LIN {X 0,Y 99.884,Z 820.994,A -85,B 0,C 180,E1 25333.007,E2 25333.007} C_VEL
LIN {X 0,Y 124.493,Z 808.852,A -85,B 0,C 180,E1 25348.353,E2 25348.353} C_VEL
LIN {X 0,Y 153.117,Z 791.255,A -85,B 0,C 180,E1 25357.972,E2 25357.972} C_VEL
LIN {X 0,Y 182.881,Z 767.638,A -85,B 0,C 180,E1 25364.239,E2 25364.239} C_VEL
LIN {X 0,Y 189.802,Z 761.231,A -85,B 0,C 180,E1 25365.397,E2 25365.397} C_VEL
LIN {X 0,Y 195.132,Z 755.346,A -85,B 0,C 180,E1 25367.364,E2 25367.364} C_VEL
LIN {X 0,Y 198.666,Z 750.355,A -85,B 0,C 180,E1 25371.032,E2 25371.032} C_VEL
LIN {X 0,Y 200.372,Z 747.755,A -85,B 0,C 180,E1 25375.668,E2 25375.668} C_VEL
LIN {X 0,Y 200.976,Z 747.527,A -85,B 0,C 180,E1 25380.001,E2 25380.001} C_VEL
LIN {X 0,Y 199.237,Z 751.38,A -85,B 0,C 180,E1 25385.39,E2 25385.39} C_VEL
LIN {X 0,Y 197.973,Z 753.101,A -85,B 0,C 180,E1 25386.177,E2 25386.177} C_VEL
LIN {X 0,Y 169.301,Z 779.906,A -85,B 0,C 180,E1 25390.356,E2 25390.356} C_VEL
LIN {X 0,Y 138.614,Z 802.307,A -85,B 0,C 180,E1 25397.113,E2 25397.113} C_VEL
LIN {X 0,Y 110.818,Z 818.489,A -85,B 0,C 180,E1 25407.373,E2 25407.373} C_VEL
LIN {X 0,Y 86.48,Z 830.411,A -85,B 0,C 180,E1 25425.552,E2 25425.552} C_VEL
LIN {X 0,Y 75.414,Z 835.837,A -85,B 0,C 180,E1 25446.328,E2 25446.328} C_VEL
LIN {X 0,Y 73.158,Z 837.803,A -85,B 0,C 180,E1 25470.002,E2 25470.002} C_VEL
LIN {X 0,Y 75.424,Z 835.865,A -85,B 0,C 180,E1 25493.673,E2 25493.673} C_VEL
LIN {X 0,Y 91.541,Z 828.062,A -85,B 0,C 180,E1 25519.694,E2 25519.694} C_VEL
LIN {X 0,Y 116.651,Z 815.401,A -85,B 0,C 180,E1 25535.309,E2 25535.309} C_VEL
LIN {X 0,Y 147.138,Z 796.73,A -85,B 0,C 180,E1 25545.104,E2 25545.104} C_VEL
LIN {X 0,Y 177.618,Z 773.044,A -85,B 0,C 180,E1 25551.026,E2 25551.026} C_VEL
LIN {X 0,Y 197.983,Z 753.354,A -85,B 0,C 180,E1 25553.813,E2 25553.813} C_VEL
LIN {X 0,Y 199.783,Z 750.548,A -85,B 0,C 180,E1 25555.653,E2 25555.653} C_VEL
LIN {X 0,Y 201.058,Z 747.717,A -85,B 0,C 180,E1 25559.999,E2 25559.999} C_VEL
LIN {X 0,Y 200.407,Z 748.005,A -85,B 0,C 180,E1 25564.332,E2 25564.332} C_VEL
LIN {X 0,Y 197.938,Z 751.928,A -85,B 0,C 180,E1 25570.415,E2 25570.415} C_VEL
LIN {X 0,Y 193.785,Z 756.272,A -85,B 0,C 180,E1 25571.361,E2 25571.361} C_VEL
LIN {X 0,Y 164.984,Z 781.309,A -85,B 0,C 180,E1 25575.978,E2 25575.978} C_VEL
LIN {X 0,Y 134.949,Z 801.449,A -85,B 0,C 180,E1 25583.231,E2 25583.231} C_VEL
LIN {X 0,Y 105.987,Z 816.488,A -85,B 0,C 180,E1 25595.339,E2 25595.339} C_VEL
LIN {X 0,Y 82.666,Z 826.048,A -85,B 0,C 180,E1 25616.668,E2 25616.668} C_VEL
LIN {X 0,Y 74.295,Z 829.174,A -85,B 0,C 180,E1 25638.239,E2 25638.239} C_VEL
LIN {X 0,Y 73.683,Z 829.562,A -85,B 0,C 180,E1 25649.998,E2 25649.998} C_VEL
LIN {X 0,Y 77.339,Z 827.963,A -85,B 0,C 180,E1 25673.048,E2 25673.048} C_VEL
LIN {X 0,Y 94.189,Z 821.445,A -85,B 0,C 180,E1 25696.33,E2 25696.33} C_VEL
LIN {X 0,Y 120.489,Z 809.306,A -85,B 0,C 180,E1 25711.593,E2 25711.593} C_VEL
LIN {X 0,Y 150.297,Z 791.716,A -85,B 0,C 180,E1 25720.803,E2 25720.803} C_VEL
LIN {X 0,Y 180.886,Z 768.123,A -85,B 0,C 180,E1 25726.661,E2 25726.661} C_VEL
LIN {X 0,Y 197.67,Z 752.007,A -85,B 0,C 180,E1 25729.325,E2 25729.325} C_VEL
LIN {X 0,Y 198.666,Z 750.355,A -85,B 0,C 180,E1 25731.032,E2 25731.032} C_VEL
LIN {X 0,Y 198.812,Z 749.478,A -85,B 0,C 180,E1 25734.15,E2 25734.15} C_VEL
LIN {X 0,Y 194.974,Z 753.929,A -85,B 0,C 180,E1 25741.229,E2 25741.229} C_VEL
LIN {X 0,Y 194.065,Z 755.858,A -85,B 0,C 180,E1 25743.982,E2 25743.982} C_VEL
LIN {X 0,Y 163.979,Z 782.599,A -85,B 0,C 180,E1 25748.268,E2 25748.268} C_VEL
LIN {X 0,Y 133.056,Z 803.862,A -85,B 0,C 180,E1 25754.716,E2 25754.716} C_VEL
LIN {X 0,Y 104.295,Z 819.434,A -85,B 0,C 180,E1 25764.867,E2 25764.867} C_VEL
LIN {X 0,Y 80.849,Z 829.952,A -85,B 0,C 180,E1 25781.493,E2 25781.493} C_VEL
LIN {X 0,Y 68.087,Z 835.382,A -85,B 0,C 180,E1 25803.596,E2 25803.596} C_VEL
LIN {X 0,Y 65.227,Z 837.358,A -85,B 0,C 180,E1 25830.002,E2 25830.002} C_VEL
LIN {X 0,Y 68.642,Z 835.155,A -85,B 0,C 180,E1 25858.083,E2 25858.083} C_VEL
LIN {X 0,Y 86.807,Z 827.462,A -85,B 0,C 180,E1 25884.111,E2 25884.111} C_VEL
LIN {X 0,Y 115.581,Z 813.857,A -85,B 0,C 180,E1 25899.888,E2 25899.888} C_VEL
LIN {X 0,Y 148.967,Z 793.752,A -85,B 0,C 180,E1 25909.005,E2 25909.005} C_VEL
LIN {X 0,Y 178.898,Z 770.432,A -85,B 0,C 180,E1 25913.957,E2 25913.957} C_VEL
LIN {X 0,Y 194.078,Z 756.16,A -85,B 0,C 180,E1 25915.86,E2 25915.86} C_VEL
LIN {X 0,Y 195.432,Z 753.425,A -85,B 0,C 180,E1 25919.999,E2 25919.999} C_VEL
LIN {X 0,Y 194.735,Z 753.771,A -85,B 0,C 180,E1 25924.458,E2 25924.458} C_VEL
LIN {X 0,Y 193.418,Z 755.527,A -85,B 0,C 180,E1 25927.98,E2 25927.98} C_VEL
LIN {X 0,Y 192.198,Z 756.934,A -85,B 0,C 180,E1 25929.063,E2 25929.063} C_VEL
LIN {X 0,Y 162.977,Z 781.775,A -85,B 0,C 180,E1 25933.293,E2 25933.293} C_VEL
LIN {X 0,Y 132.746,Z 801.47,A -85,B 0,C 180,E1 25939.833,E2 25939.833} C_VEL
LIN {X 0,Y 103.062,Z 816.261,A -85,B 0,C 180,E1 25950.873,E2 25950.873} C_VEL
LIN {X 0,Y 77.793,Z 825.982,A -85,B 0,C 180,E1 25971.115,E2 25971.115} C_VEL
LIN {X 0,Y 66.554,Z 829.618,A -85,B 0,C 180,E1 25996.848,E2 25996.848} C_VEL
LIN {X 0,Y 65.782,Z 830.006,A -85,B 0,C 180,E1 26009.998,E2 26009.998} C_VEL
LIN {X 0,Y 70.094,Z 828.41,A -85,B 0,C 180,E1 26035.592,E2 26035.592} C_VEL
LIN {X 0,Y 84.222,Z 823.666,A -85,B 0,C 180,E1 26055.975,E2 26055.975} C_VEL
LIN {X 0,Y 110.809,Z 812.725,A -85,B 0,C 180,E1 26072.637,E2 26072.637} C_VEL
LIN {X 0,Y 139.683,Z 797.315,A -85,B 0,C 180,E1 26081.877,E2 26081.877} C_VEL
LIN {X 0,Y 170.365,Z 775.928,A -85,B 0,C 180,E1 26087.84,E2 26087.84} C_VEL
LIN {X 0,Y 192.711,Z 756.183,A -85,B 0,C 180,E1 26090.961,E2 26090.961} C_VEL
LIN {X 0,Y 194.716,Z 753.505,A -85,B 0,C 180,E1 26095.541,E2 26095.541} C_VEL
LIN {X 0,Y 195.349,Z 753.236,A -85,B 0,C 180,E1 26100.001,E2 26100.001} C_VEL
LIN {X 0,Y 194.974,Z 753.929,A -85,B 0,C 180,E1 26101.229,E2 26101.229} C_VEL
LIN {X 0,Y 192.253,Z 756.976,A -85,B 0,C 180,E1 26102.508,E2 26102.508} C_VEL
LIN {X 0,Y 178.528,Z 769.454,A -85,B 0,C 180,E1 26103.404,E2 26103.404} C_VEL
LIN {X 0,Y 147.135,Z 793.447,A -85,B 0,C 180,E1 26107.939,E2 26107.939} C_VEL
LIN {X 0,Y 113.771,Z 812.934,A -85,B 0,C 180,E1 26115.967,E2 26115.967} C_VEL
LIN {X 0,Y 83.388,Z 826.508,A -85,B 0,C 180,E1 26130.412,E2 26130.412} C_VEL
LIN {X 0,Y 63.672,Z 833.955,A -85,B 0,C 180,E1 26153.528,E2 26153.528} C_VEL
LIN {X 0,Y 57.593,Z 836.355,A -85,B 0,C 180,E1 26174.761,E2 26174.761} C_VEL
LIN {X 0,Y 57.315,Z 836.914,A -85,B 0,C 180,E1 26190.003,E2 26190.003} C_VEL
LIN {X 0,Y 60.982,Z 834.96,A -85,B 0,C 180,E1 26219.775,E2 26219.775} C_VEL
LIN {X 0,Y 80.731,Z 827.598,A -85,B 0,C 180,E1 26247.563,E2 26247.563} C_VEL
LIN {X 0,Y 110.792,Z 814.475,A -85,B 0,C 180,E1 26263.063,E2 26263.063} C_VEL
LIN {X 0,Y 145.353,Z 794.817,A -85,B 0,C 180,E1 26271.721,E2 26271.721} C_VEL
LIN {X 0,Y 178.223,Z 769.94,A -85,B 0,C 180,E1 26276.57,E2 26276.57} C_VEL
LIN {X 0,Y 188.15,Z 760.95,A -85,B 0,C 180,E1 26277.649,E2 26277.649} C_VEL
LIN {X 0,Y 189.628,Z 758.959,A -85,B 0,C 180,E1 26279.999,E2 26279.999} C_VEL
LIN {X 0,Y 188.288,Z 759.942,A -85,B 0,C 180,E1 26286.01,E2 26286.01} C_VEL
LIN {X 0,Y 187.946,Z 760.382,A -85,B 0,C 180,E1 26286.89,E2 26286.89} C_VEL
LIN {X 0,Y 158.206,Z 784.528,A -85,B 0,C 180,E1 26291.033,E2 26291.033} C_VEL
LIN {X 0,Y 126.907,Z 803.793,A -85,B 0,C 180,E1 26297.359,E2 26297.359} C_VEL
LIN {X 0,Y 97.209,Z 817.544,A -85,B 0,C 180,E1 26307.852,E2 26307.852} C_VEL
LIN {X 0,Y 69.899,Z 826.939,A -85,B 0,C 180,E1 26329.469,E2 26329.469} C_VEL
LIN {X 0,Y 58.861,Z 830.063,A -85,B 0,C 180,E1 26355.092,E2 26355.092} C_VEL
LIN {X 0,Y 57.899,Z 830.448,A -85,B 0,C 180,E1 26369.997,E2 26369.997} C_VEL
LIN {X 0,Y 63.019,Z 828.857,A -85,B 0,C 180,E1 26398.716,E2 26398.716} C_VEL
LIN {X 0,Y 78.876,Z 824.114,A -85,B 0,C 180,E1 26420.155,E2 26420.155} C_VEL
LIN {X 0,Y 107.374,Z 813.178,A -85,B 0,C 180,E1 26436.422,E2 26436.422} C_VEL
LIN {X 0,Y 138.883,Z 796.875,A -85,B 0,C 180,E1 26445.352,E2 26445.352} C_VEL
LIN {X 0,Y 170.667,Z 774.971,A -85,B 0,C 180,E1 26450.723,E2 26450.723} C_VEL
LIN {X 0,Y 187.837,Z 760.224,A -85,B 0,C 180,E1 26453.064,E2 26453.064} C_VEL
LIN {X 0,Y 188.833,Z 759.063,A -85,B 0,C 180,E1 26455.402,E2 26455.402} C_VEL
LIN {X 0,Y 189.277,Z 759.221,A -85,B 0,C 180,E1 26460.822,E2 26460.822} C_VEL
LIN {X 0,Y 188.874,Z 759.929,A -85,B 0,C 180,E1 26462.014,E2 26462.014} C_VEL
LIN {X 0,Y 178.528,Z 769.454,A -85,B 0,C 180,E1 26463.404,E2 26463.404} C_VEL
LIN {X 0,Y 164.754,Z 780.338,A -85,B 0,C 180,E1 26463.71,E2 26463.71} C_VEL
LIN {X 0,Y 150.338,Z 790.211,A -85,B 0,C 180,E1 26464.149,E2 26464.149} C_VEL
LIN {X 0,Y 118.789,Z 808.908,A -85,B 0,C 180,E1 26470.089,E2 26470.089} C_VEL
LIN {X 0,Y 86.351,Z 823.488,A -85,B 0,C 180,E1 26481.504,E2 26481.504} C_VEL
LIN {X 0,Y 61.326,Z 832.18,A -85,B 0,C 180,E1 26502.216,E2 26502.216} C_VEL
LIN {X 0,Y 49.906,Z 835.905,A -85,B 0,C 180,E1 26532.343,E2 26532.343} C_VEL
LIN {X 0,Y 49.374,Z 836.468,A -85,B 0,C 180,E1 26550.003,E2 26550.003} C_VEL
LIN {X 0,Y 54.102,Z 834.506,A -85,B 0,C 180,E1 26584.039,E2 26584.039} C_VEL
LIN {X 0,Y 76.643,Z 827.139,A -85,B 0,C 180,E1 26612.748,E2 26612.748} C_VEL
LIN {X 0,Y 108.684,Z 814.011,A -85,B 0,C 180,E1 26627.207,E2 26627.207} C_VEL
LIN {X 0,Y 144.395,Z 794.344,A -85,B 0,C 180,E1 26634.963,E2 26634.963} C_VEL
LIN {X 0,Y 177.921,Z 769.447,A -85,B 0,C 180,E1 26639.192,E2 26639.192} C_VEL
LIN {X 0,Y 183.698,Z 764.39,A -85,B 0,C 180,E1 26639.999,E2 26639.999} C_VEL
LIN {X 0,Y 182.421,Z 765.109,A -85,B 0,C 180,E1 26645.136,E2 26645.136} C_VEL
LIN {X 0,Y 151.362,Z 788.656,A -85,B 0,C 180,E1 26648.958,E2 26648.958} C_VEL
LIN {X 0,Y 119.97,Z 806.58,A -85,B 0,C 180,E1 26654.969,E2 26654.969} C_VEL
LIN {X 0,Y 89.506,Z 819.481,A -85,B 0,C 180,E1 26665.441,E2 26665.441} C_VEL
LIN {X 0,Y 63.06,Z 827.637,A -85,B 0,C 180,E1 26686.07,E2 26686.07} C_VEL
LIN {X 0,Y 51.239,Z 830.508,A -85,B 0,C 180,E1 26712.81,E2 26712.81} C_VEL
LIN {X 0,Y 49.995,Z 830.892,A -85,B 0,C 180,E1 26729.997,E2 26729.997} C_VEL
LIN {X 0,Y 56.175,Z 829.304,A -85,B 0,C 180,E1 26762.615,E2 26762.615} C_VEL
LIN {X 0,Y 79.545,Z 822.796,A -85,B 0,C 180,E1 26788.924,E2 26788.924} C_VEL
LIN {X 0,Y 111.095,Z 810.662,A -85,B 0,C 180,E1 26802.547,E2 26802.547} C_VEL
LIN {X 0,Y 144.205,Z 793.094,A -85,B 0,C 180,E1 26809.831,E2 26809.831} C_VEL
LIN {X 0,Y 176.909,Z 769.579,A -85,B 0,C 180,E1 26814.206,E2 26814.206} C_VEL
LIN {X 0,Y 182.434,Z 764.862,A -85,B 0,C 180,E1 26814.8,E2 26814.8} C_VEL
LIN {X 0,Y 183.63,Z 764.22,A -85,B 0,C 180,E1 26820.001,E2 26820.001} C_VEL
LIN {X 0,Y 154.352,Z 787.527,A -85,B 0,C 180,E1 26823.593,E2 26823.593} C_VEL
LIN {X 0,Y 150.338,Z 790.211,A -85,B 0,C 180,E1 26824.149,E2 26824.149} C_VEL
LIN {X 0,Y 135.405,Z 799.256,A -85,B 0,C 180,E1 26824.822,E2 26824.822} C_VEL
LIN {X 0,Y 119.946,Z 807.298,A -85,B 0,C 180,E1 26825.703,E2 26825.703} C_VEL
LIN {X 0,Y 87.793,Z 821.536,A -85,B 0,C 180,E1 26834.544,E2 26834.544} C_VEL
LIN {X 0,Y 56.17,Z 831.722,A -85,B 0,C 180,E1 26856.041,E2 26856.041} C_VEL
LIN {X 0,Y 42.343,Z 835.455,A -85,B 0,C 180,E1 26889.053,E2 26889.053} C_VEL
LIN {X 0,Y 41.429,Z 836.022,A -85,B 0,C 180,E1 26910.004,E2 26910.004} C_VEL
LIN {X 0,Y 47.607,Z 834.052,A -85,B 0,C 180,E1 26949.503,E2 26949.503} C_VEL
LIN {X 0,Y 73.26,Z 826.68,A -85,B 0,C 180,E1 26978.441,E2 26978.441} C_VEL
LIN {X 0,Y 107.169,Z 813.551,A -85,B 0,C 180,E1 26991.48,E2 26991.48} C_VEL
LIN {X 0,Y 143.908,Z 793.875,A -85,B 0,C 180,E1 26998.211,E2 26998.211} C_VEL
LIN {X 0,Y 177.143,Z 769.661,A -85,B 0,C 180,E1 27001.946,E2 27001.946} C_VEL
LIN {X 0,Y 176.977,Z 769.732,A -85,B 0,C 180,E1 27002.843,E2 27002.843} C_VEL
LIN {X 0,Y 146.656,Z 791.472,A -85,B 0,C 180,E1 27006.441,E2 27006.441} C_VEL
LIN {X 0,Y 111.616,Z 810.098,A -85,B 0,C 180,E1 27012.672,E2 27012.672} C_VEL
LIN {X 0,Y 81.99,Z 821.425,A -85,B 0,C 180,E1 27022.58,E2 27022.58} C_VEL
LIN {X 0,Y 58.698,Z 827.831,A -85,B 0,C 180,E1 27039.298,E2 27039.298} C_VEL
LIN {X 0,Y 43.725,Z 830.953,A -85,B 0,C 180,E1 27069.737,E2 27069.737} C_VEL
LIN {X 0,Y 42.117,Z 831.334,A -85,B 0,C 180,E1 27089.996,E2 27089.996} C_VEL
LIN {X 0,Y 49.663,Z 829.75,A -85,B 0,C 180,E1 27127.566,E2 27127.566} C_VEL
LIN {X 0,Y 75.728,Z 823.244,A -85,B 0,C 180,E1 27154.113,E2 27154.113} C_VEL
LIN {X 0,Y 108.963,Z 811.114,A -85,B 0,C 180,E1 27166.564,E2 27166.564} C_VEL
LIN {X 0,Y 143.013,Z 793.554,A -85,B 0,C 180,E1 27172.974,E2 27172.974} C_VEL
LIN {X 0,Y 176.924,Z 769.531,A -85,B 0,C 180,E1 27176.935,E2 27176.935} C_VEL
LIN {X 0,Y 177.12,Z 769.448,A -85,B 0,C 180,E1 27178.061,E2 27178.061} C_VEL
LIN {X 0,Y 145.778,Z 792.49,A -85,B 0,C 180,E1 27181.55,E2 27181.55} C_VEL
LIN {X 0,Y 119.946,Z 807.298,A -85,B 0,C 180,E1 27185.703,E2 27185.703} C_VEL
LIN {X 0,Y 104.006,Z 814.363,A -85,B 0,C 180,E1 27186.888,E2 27186.888} C_VEL
LIN {X 0,Y 87.86,Z 820.433,A -85,B 0,C 180,E1 27188.679,E2 27188.679} C_VEL
LIN {X 0,Y 55.766,Z 830.347,A -85,B 0,C 180,E1 27205.007,E2 27205.007} C_VEL
LIN {X 0,Y 34.963,Z 835.004,A -85,B 0,C 180,E1 27244.344,E2 27244.344} C_VEL
LIN {X 0,Y 33.48,Z 835.576,A -85,B 0,C 180,E1 27270.005,E2 27270.005} C_VEL
LIN {X 0,Y 41.673,Z 833.597,A -85,B 0,C 180,E1 27316.611,E2 27316.611} C_VEL
LIN {X 0,Y 70.665,Z 826.221,A -85,B 0,C 180,E1 27344.623,E2 27344.623} C_VEL
LIN {X 0,Y 106.266,Z 813.092,A -85,B 0,C 180,E1 27355.845,E2 27355.845} C_VEL
LIN {X 0,Y 141.98,Z 794.533,A -85,B 0,C 180,E1 27361.264,E2 27361.264} C_VEL
LIN {X 0,Y 151.522,Z 788.479,A -85,B 0,C 180,E1 27362.221,E2 27362.221} C_VEL
LIN {X 0,Y 151.58,Z 788.402,A -85,B 0,C 180,E1 27362.727,E2 27362.727} C_VEL
LIN {X 0,Y 117.97,Z 806.976,A -85,B 0,C 180,E1 27367.181,E2 27367.181} C_VEL
LIN {X 0,Y 84.722,Z 820.114,A -85,B 0,C 180,E1 27375.246,E2 27375.246} C_VEL
LIN {X 0,Y 54.003,Z 828.279,A -85,B 0,C 180,E1 27392.738,E2 27392.738} C_VEL
LIN {X 0,Y 36.387,Z 831.398,A -85,B 0,C 180,E1 27425.407,E2 27425.407} C_VEL
LIN {X 0,Y 34.211,Z 831.777,A -85,B 0,C 180,E1 27449.995,E2 27449.995} C_VEL
LIN {X 0,Y 49.061,Z 829.257,A -85,B 0,C 180,E1 27501.894,E2 27501.894} C_VEL
LIN {X 0,Y 79.278,Z 821.786,A -85,B 0,C 180,E1 27522.719,E2 27522.719} C_VEL
LIN {X 0,Y 115.625,Z 807.932,A -85,B 0,C 180,E1 27532.303,E2 27532.303} C_VEL
LIN {X 0,Y 149.716,Z 789.397,A -85,B 0,C 180,E1 27536.991,E2 27536.991} C_VEL
LIN {X 0,Y 151.587,Z 788.215,A -85,B 0,C 180,E1 27537.17,E2 27537.17} C_VEL
LIN {X 0,Y 151.517,Z 788.308,A -85,B 0,C 180,E1 27537.772,E2 27537.772} C_VEL
LIN {X 0,Y 117.415,Z 807.794,A -85,B 0,C 180,E1 27542.097,E2 27542.097} C_VEL
LIN {X 0,Y 87.86,Z 820.433,A -85,B 0,C 180,E1 27548.679,E2 27548.679} C_VEL
LIN {X 0,Y 71.428,Z 825.402,A -85,B 0,C 180,E1 27551.301,E2 27551.301} C_VEL
LIN {X 0,Y 54.972,Z 829.347,A -85,B 0,C 180,E1 27555.526,E2 27555.526} C_VEL
LIN {X 0,Y 36.572,Z 833.111,A -85,B 0,C 180,E1 27574.115,E2 27574.115} C_VEL
LIN {X 0,Y 25.543,Z 835.131,A -85,B 0,C 180,E1 27630.006,E2 27630.006} C_VEL
LIN {X 0,Y 36.578,Z 833.142,A -85,B 0,C 180,E1 27685.886,E2 27685.886} C_VEL
LIN {X 0,Y 68.944,Z 825.763,A -85,B 0,C 180,E1 27711.213,E2 27711.213} C_VEL
LIN {X 0,Y 105.988,Z 812.629,A -85,B 0,C 180,E1 27720.293,E2 27720.293} C_VEL
LIN {X 0,Y 121.232,Z 805.647,A -85,B 0,C 180,E1 27722.385,E2 27722.385} C_VEL
LIN {X 0,Y 121.271,Z 805.598,A -85,B 0,C 180,E1 27722.79,E2 27722.79} C_VEL
LIN {X 0,Y 84.506,Z 820.095,A -85,B 0,C 180,E1 27729.517,E2 27729.517} C_VEL
LIN {X 0,Y 50.132,Z 828.727,A -85,B 0,C 180,E1 27745.029,E2 27745.029} C_VEL
LIN {X 0,Y 29.359,Z 831.843,A -85,B 0,C 180,E1 27778.949,E2 27778.949} C_VEL
LIN {X 0,Y 26.303,Z 832.221,A -85,B 0,C 180,E1 27809.994,E2 27809.994} C_VEL
LIN {X 0,Y 38.312,Z 830.641,A -85,B 0,C 180,E1 27862.214,E2 27862.214} C_VEL
LIN {X 0,Y 70.232,Z 824.144,A -85,B 0,C 180,E1 27885.944,E2 27885.944} C_VEL
LIN {X 0,Y 106.392,Z 812.021,A -85,B 0,C 180,E1 27894.959,E2 27894.959} C_VEL
LIN {X 0,Y 121.272,Z 805.463,A -85,B 0,C 180,E1 27897.142,E2 27897.142} C_VEL
LIN {X 0,Y 121.225,Z 805.522,A -85,B 0,C 180,E1 27897.634,E2 27897.634} C_VEL
LIN {X 0,Y 84.902,Z 820.698,A -85,B 0,C 180,E1 27903.833,E2 27903.833} C_VEL
LIN {X 0,Y 54.972,Z 829.347,A -85,B 0,C 180,E1 27915.526,E2 27915.526} C_VEL
LIN {X 0,Y 42.942,Z 831.639,A -85,B 0,C 180,E1 27921.185,E2 27921.185} C_VEL
LIN {X 0,Y 24.915,Z 833.703,A -85,B 0,C 180,E1 27935.72,E2 27935.72} C_VEL
LIN {X 0,Y 23.407,Z 833.85,A -85,B 0,C 180,E1 27939.523,E2 27939.523} C_VEL
LIN {X 0,Y 17.584,Z 834.684,A -85,B 0,C 180,E1 27990.009,E2 27990.009} C_VEL
LIN {X 0,Y 32.734,Z 832.69,A -85,B 0,C 180,E1 28057.692,E2 28057.692} C_VEL
LIN {X 0,Y 68.175,Z 825.304,A -85,B 0,C 180,E1 28078.036,E2 28078.036} C_VEL
LIN {X 0,Y 90.951,Z 818.151,A -85,B 0,C 180,E1 28082.753,E2 28082.753} C_VEL
LIN {X 0,Y 54.308,Z 827.907,A -85,B 0,C 180,E1 28092.625,E2 28092.625} C_VEL
LIN {X 0,Y 22.93,Z 832.288,A -85,B 0,C 180,E1 28128.669,E2 28128.669} C_VEL
LIN {X 0,Y 18.395,Z 832.665,A -85,B 0,C 180,E1 28169.991,E2 28169.991} C_VEL
LIN {X 0,Y 36.281,Z 830.803,A -85,B 0,C 180,E1 28235.341,E2 28235.341} C_VEL
LIN {X 0,Y 68.729,Z 824.594,A -85,B 0,C 180,E1 28252.428,E2 28252.428} C_VEL
LIN {X 0,Y 90.942,Z 818.059,A -85,B 0,C 180,E1 28257.282,E2 28257.282} C_VEL
LIN {X 0,Y 51.361,Z 829.332,A -85,B 0,C 180,E1 28267.941,E2 28267.941} C_VEL
LIN {X 0,Y 23.407,Z 833.85,A -85,B 0,C 180,E1 28299.523,E2 28299.523} C_VEL
LIN {X 0,Y 14.939,Z 834.532,A -85,B 0,C 180,E1 28330.471,E2 28330.471} C_VEL
LIN {X 0,Y 18.051,Z 833.537,A -85,B 0,C 180,E1 28416.618,E2 28416.618} C_VEL
LIN {X 0,Y 46.964,Z 829.669,A -85,B 0,C 180,E1 28439.997,E2 28439.997} C_VEL
LIN {X 0,Y 56.525,Z 827.709,A -85,B 0,C 180,E1 28442.654,E2 28442.654} C_VEL
LIN {X 0,Y 31.206,Z 831.571,A -85,B 0,C 180,E1 28453.965,E2 28453.965} C_VEL
LIN {X 0,Y 10.496,Z 833.108,A -85,B 0,C 180,E1 28529.984,E2 28529.984} C_VEL
LIN {X 0,Y 31.212,Z 831.534,A -85,B 0,C 180,E1 28605.95,E2 28605.95} C_VEL
LIN {X 0,Y 56.649,Z 827.623,A -85,B 0,C 180,E1 28617.317,E2 28617.317} C_VEL
LIN {X 0,Y 30.581,Z 832.201,A -85,B 0,C 180,E1 28628.066,E2 28628.066} C_VEL
LIN {X 0,Y 9.643,Z 834.238,A -85,B 0,C 180,E1 28710.017,E2 28710.017} C_VEL
LIN {X 0,Y 18.051,Z 833.537,A -85,B 0,C 180,E1 28776.618,E2 28776.618} C_VEL
LIN {X 0,Y 14.146,Z 833.507,A -85,B 0,C 180,E1 28788.096,E2 28788.096} C_VEL
LIN {X 0,Y 2.205,Z 833.569,A -85,B 0,C 180,E1 28909.108,E2 28909.108} C_VEL
LIN {X 0,Y 5.438,Z 833.422,A -85,B 0,C 180,E1 28956.094,E2 28956.094} C_VEL
LIN {X 0,Y 15.204,Z 833.155,A -85,B 0,C 180,E1 28974.629,E2 28974.629} C_VEL
LIN {X 0,Y 1.672,Z 833.791,A -85,B 0,C 180,E1 29070.097,E2 29070.097} C_VEL
LIN {X 0,Y 15.204,Z 833.178,A -85,B 0,C 180,E1 29165.139,E2 29165.139} C_VEL
LIN {X 0,Y 5.438,Z 833.422,A -85,B 0,C 180,E1 29316.094,E2 29316.094} C_VEL
LIN {X 0,Y 7.31,Z 835.421,A -85,B 0,C 180,E1 29323.741,E2 29323.741} C_VEL
LIN {X 0,Y 7.31,Z 862.5,A -85,B 0,C 180,E1 29323.741,E2 29323.741} C_VEL
LIN {X 0,Y 7.31,Z 862.5,A -85,B 0,C 180,E1 29323.741,E2 29323.741}

QRS_NEXT_CUT()
PTP {E1 29336.868,E2 29336.868}
PTP {X 0,Y 607.922,A -85,B 0,C 180,E1 29336.868,E2 29336.868,E3 0,E4 0,E5 0,E6 0}
QRS_SPEED_INIT()
LIN {X 0,Y 607.922,Z 862.5,A -85,B 0,C 180,E1 29336.868,E2 29336.868,E3 0,E4 0,E5 0,E6 0} C_VEL
LIN {X 0,Y 607.922,Z 262.089,A -85,B 0,C 180,E1 29336.868,E2 29336.868} C_VEL
LIN {X 0,Y 607.922,Z 254.014,A -85,B 0,C 180,E1 29336.868,E2 29336.868} C_VEL
LIN {X 0,Y 607.917,Z 252.014,A -85,B 0,C 180,E1 29336.68,E2 29336.68} C_VEL
LIN {X 0,Y 607.854,Z 252.011,A -85,B 0,C 180,E1 29333.578,E2 29333.578} C_VEL
LIN {X 0,Y 607.917,Z 252.011,A -85,B 0,C 180,E1 29330.533,E2 29330.533} C_VEL
LIN {X 0,Y 607.86,Z 252.012,A -85,B 0,C 180,E1 29327.46,E2 29327.46} C_VEL
LIN {X 0,Y 607.916,Z 252.009,A -85,B 0,C 180,E1 29324.351,E2 29324.351} C_VEL
LIN {X 0,Y 607.875,Z 252.012,A -85,B 0,C 180,E1 29321.192,E2 29321.192} C_VEL
LIN {X 0,Y 607.901,Z 252.006,A -85,B 0,C 180,E1 29317.975,E2 29317.975} C_VEL
LIN {X 0,Y 607.907,Z 252.015,A -85,B 0,C 180,E1 29314.768,E2 29314.768} C_VEL
LIN {X 0,Y 607.885,Z 252.008,A -85,B 0,C 180,E1 29311.618,E2 29311.618} C_VEL
LIN {X 0,Y 607.912,Z 252.012,A -85,B 0,C 180,E1 29308.575,E2 29308.575} C_VEL
LIN {X 0,Y 607.886,Z 252.009,A -85,B 0,C 180,E1 29305.426,E2 29305.426} C_VEL
LIN {X 0,Y 607.905,Z 252.01,A -85,B 0,C 180,E1 29302.395,E2 29302.395} C_VEL
LIN {X 0,Y 607.891,Z 252.01,A -85,B 0,C 180,E1 29299.233,E2 29299.233} C_VEL
LIN {X 0,Y 607.902,Z 252.008,A -85,B 0,C 180,E1 29296.087,E2 29296.087} C_VEL
LIN {X 0,Y 607.904,Z 252.012,A -85,B 0,C 180,E1 29292.915,E2 29292.915} C_VEL
LIN {X 0,Y 607.91,Z 252.004,A -85,B 0,C 180,E1 29289.654,E2 29289.654} C_VEL
LIN {X 0,Y 607.899,Z 252.013,A -85,B 0,C 180,E1 29286.423,E2 29286.423} C_VEL
LIN {X 0,Y 607.903,Z 252.007,A -85,B 0,C 180,E1 29283.209,E2 29283.209} C_VEL
LIN {X 0,Y 607.908,Z 252.244,A -85,B 0,C 180,E1 29282.871,E2 29282.871} C_VEL
LIN {X 0,Y 607.916,Z 262.06,A -85,B 0,C 180,E1 29282.155,E2 29282.155} C_VEL
LIN {X 0,Y 607.91,Z 307.319,A -85,B 0,C 180,E1 29279.079,E2 29279.079} C_VEL
LIN {X 0,Y 607.915,Z 329.228,A -85,B 0,C 180,E1 29277.639,E2 29277.639} C_VEL
LIN {X 0,Y 607.906,Z 572.151,A -85,B 0,C 180,E1 29274.503,E2 29274.503} C_VEL
LIN {X 0,Y 607.916,Z 596.076,A -85,B 0,C 180,E1 29274.138,E2 29274.138} C_VEL
LIN {X 0,Y 607.907,Z 615.328,A -85,B 0,C 180,E1 29273.686,E2 29273.686} C_VEL
LIN {X 0,Y 607.906,Z 635.144,A -85,B 0,C 180,E1 29273.044,E2 29273.044} C_VEL
LIN {X 0,Y 607.914,Z 653.488,A -85,B 0,C 180,E1 29272.278,E2 29272.278} C_VEL
LIN {X 0,Y 607.918,Z 672.334,A -85,B 0,C 180,E1 29271.314,E2 29271.314} C_VEL
LIN {X 0,Y 607.918,Z 690.309,A -85,B 0,C 180,E1 29270.205,E2 29270.205} C_VEL
LIN {X 0,Y 607.912,Z 707.273,A -85,B 0,C 180,E1 29268.963,E2 29268.963} C_VEL
LIN {X 0,Y 607.916,Z 723.45,A -85,B 0,C 180,E1 29267.566,E2 29267.566} C_VEL
LIN {X 0,Y 607.913,Z 738.451,A -85,B 0,C 180,E1 29266.04,E2 29266.04} C_VEL
LIN {X 0,Y 607.916,Z 752.426,A -85,B 0,C 180,E1 29264.361,E2 29264.361} C_VEL
LIN {X 0,Y 607.912,Z 764.497,A -85,B 0,C 180,E1 29262.635,E2 29262.635} C_VEL
LIN {X 0,Y 607.904,Z 774.619,A -85,B 0,C 180,E1 29260.903,E2 29260.903} C_VEL
LIN {X 0,Y 607.912,Z 783.37,A -85,B 0,C 180,E1 29259.084,E2 29259.084} C_VEL
LIN {X 0,Y 607.907,Z 790.348,A -85,B 0,C 180,E1 29257.276,E2 29257.276} C_VEL
LIN {X 0,Y 607.903,Z 795.888,A -85,B 0,C 180,E1 29255.379,E2 29255.379} C_VEL
LIN {X 0,Y 607.901,Z 799.664,A -85,B 0,C 180,E1 29253.489,E2 29253.489} C_VEL
LIN {X 0,Y 607.903,Z 801.841,A -85,B 0,C 180,E1 29251.602,E2 29251.602} C_VEL
LIN {X 0,Y 607.904,Z 802.45,A -85,B 0,C 180,E1 29249.717,E2 29249.717} C_VEL
LIN {X 0,Y 607.911,Z 801.498,A -85,B 0,C 180,E1 29247.832,E2 29247.832} C_VEL
LIN {X 0,Y 607.913,Z 798.71,A -85,B 0,C 180,E1 29245.85,E2 29245.85} C_VEL
LIN {X 0,Y 607.919,Z 794.356,A -85,B 0,C 180,E1 29243.958,E2 29243.958} C_VEL
LIN {X 0,Y 607.915,Z 788.287,A -85,B 0,C 180,E1 29242.059,E2 29242.059} C_VEL
LIN {X 0,Y 607.91,Z 780.817,A -85,B 0,C 180,E1 29240.247,E2 29240.247} C_VEL
LIN {X 0,Y 607.904,Z 771.474,A -85,B 0,C 180,E1 29238.425,E2 29238.425} C_VEL
LIN {X 0,Y 607.912,Z 760.614,A -85,B 0,C 180,E1 29236.688,E2 29236.688} C_VEL
LIN {X 0,Y 607.91,Z 748.345,A -85,B 0,C 180,E1 29235.036,E2 29235.036} C_VEL
LIN {X 0,Y 607.916,Z 734.67,A -85,B 0,C 180,E1 29233.469,E2 29233.469} C_VEL
LIN {X 0,Y 607.912,Z 719.508,A -85,B 0,C 180,E1 29231.989,E2 29231.989} C_VEL
LIN {X 0,Y 607.918,Z 702.707,A -85,B 0,C 180,E1 29230.596,E2 29230.596} C_VEL
LIN {X 0,Y 607.918,Z 685.576,A -85,B 0,C 180,E1 29229.393,E2 29229.393} C_VEL
LIN {X 0,Y 607.918,Z 667.445,A -85,B 0,C 180,E1 29228.322,E2 29228.322} C_VEL
LIN {X 0,Y 607.918,Z 648.751,A -85,B 0,C 180,E1 29227.416,E2 29227.416} C_VEL
LIN {X 0,Y 607.915,Z 629.645,A -85,B 0,C 180,E1 29226.674,E2 29226.674} C_VEL
LIN {X 0,Y 607.906,Z 609.883,A -85,B 0,C 180,E1 29226.082,E2 29226.082} C_VEL
LIN {X 0,Y 607.913,Z 589.981,A -85,B 0,C 180,E1 29225.657,E2 29225.657} C_VEL
LIN {X 0,Y 607.914,Z 329.113,A -85,B 0,C 180,E1 29222.267,E2 29222.267} C_VEL
LIN {X 0,Y 607.918,Z 285.168,A -85,B 0,C 180,E1 29219.338,E2 29219.338} C_VEL
LIN {X 0,Y 607.911,Z 252.36,A -85,B 0,C 180,E1 29217.059,E2 29217.059} C_VEL
LIN {X 0,Y 607.919,Z 252.003,A -85,B 0,C 180,E1 29216.454,E2 29216.454} C_VEL
LIN {X 0,Y 607.912,Z 252.014,A -85,B 0,C 180,E1 29213.108,E2 29213.108} C_VEL
LIN {X 0,Y 607.895,Z 252.006,A -85,B 0,C 180,E1 29209.977,E2 29209.977} C_VEL
LIN {X 0,Y 607.9,Z 252.01,A -85,B 0,C 180,E1 29206.827,E2 29206.827} C_VEL
LIN {X 0,Y 607.896,Z 252.01,A -85,B 0,C 180,E1 29203.694,E2 29203.694} C_VEL
LIN {X 0,Y 607.897,Z 252.007,A -85,B 0,C 180,E1 29200.518,E2 29200.518} C_VEL
LIN {X 0,Y 607.907,Z 252.013,A -85,B 0,C 180,E1 29197.367,E2 29197.367} C_VEL
LIN {X 0,Y 607.914,Z 252.004,A -85,B 0,C 180,E1 29194.115,E2 29194.115} C_VEL
LIN {X 0,Y 607.89,Z 252.011,A -85,B 0,C 180,E1 29190.845,E2 29190.845} C_VEL
LIN {X 0,Y 607.909,Z 252.007,A -85,B 0,C 180,E1 29187.74,E2 29187.74} C_VEL
LIN {X 0,Y 607.879,Z 252.01,A -85,B 0,C 180,E1 29184.555,E2 29184.555} C_VEL
LIN {X 0,Y 607.912,Z 252.012,A -85,B 0,C 180,E1 29181.416,E2 29181.416} C_VEL
LIN {X 0,Y 607.876,Z 252.009,A -85,B 0,C 180,E1 29178.311,E2 29178.311} C_VEL
LIN {X 0,Y 607.899,Z 252.014,A -85,B 0,C 180,E1 29175.063,E2 29175.063} C_VEL
LIN {X 0,Y 607.887,Z 252.008,A -85,B 0,C 180,E1 29171.961,E2 29171.961} C_VEL
LIN {X 0,Y 607.867,Z 252.013,A -85,B 0,C 180,E1 29168.704,E2 29168.704} C_VEL
LIN {X 0,Y 607.91,Z 252.008,A -85,B 0,C 180,E1 29165.664,E2 29165.664} C_VEL
LIN {X 0,Y 607.855,Z 252.012,A -85,B 0,C 180,E1 29162.546,E2 29162.546} C_VEL
LIN {X 0,Y 607.912,Z 252.01,A -85,B 0,C 180,E1 29159.529,E2 29159.529} C_VEL
LIN {X 0,Y 607.845,Z 252.013,A -85,B 0,C 180,E1 29156.416,E2 29156.416} C_VEL
LIN {X 0,Y 607.911,Z 252.013,A -85,B 0,C 180,E1 29153.389,E2 29153.389} C_VEL
LIN {X 0,Y 607.835,Z 252.014,A -85,B 0,C 180,E1 29150.341,E2 29150.341} C_VEL
LIN {X 0,Y 607.918,Z 252.014,A -85,B 0,C 180,E1 29147.268,E2 29147.268} C_VEL
LIN {X 0,Y 607.826,Z 252.015,A -85,B 0,C 180,E1 29144.214,E2 29144.214} C_VEL
LIN {X 0,Y 607.906,Z 252.015,A -85,B 0,C 180,E1 29141.194,E2 29141.194} C_VEL
LIN {X 0,Y 607.835,Z 252.014,A -85,B 0,C 180,E1 29138.176,E2 29138.176} C_VEL
LIN {X 0,Y 607.919,Z 252.012,A -85,B 0,C 180,E1 29135.099,E2 29135.099} C_VEL
LIN {X 0,Y 607.845,Z 252.013,A -85,B 0,C 180,E1 29132.043,E2 29132.043} C_VEL
LIN {X 0,Y 607.903,Z 252.01,A -85,B 0,C 180,E1 29128.905,E2 29128.905} C_VEL
LIN {X 0,Y 607.857,Z 252.013,A -85,B 0,C 180,E1 29125.882,E2 29125.882} C_VEL
LIN {X 0,Y 607.902,Z 252.008,A -85,B 0,C 180,E1 29122.752,E2 29122.752} C_VEL
LIN {X 0,Y 607.87,Z 252.013,A -85,B 0,C 180,E1 29119.727,E2 29119.727} C_VEL
LIN {X 0,Y 607.882,Z 252.009,A -85,B 0,C 180,E1 29116.435,E2 29116.435} C_VEL
LIN {X 0,Y 607.908,Z 252.014,A -85,B 0,C 180,E1 29113.302,E2 29113.302} C_VEL
LIN {X 0,Y 607.874,Z 252.01,A -85,B 0,C 180,E1 29110.106,E2 29110.106} C_VEL
LIN {X 0,Y 607.911,Z 252.003,A -85,B 0,C 180,E1 29107.01,E2 29107.01} C_VEL
LIN {X 0,Y 607.897,Z 252.254,A -85,B 0,C 180,E1 29105.463,E2 29105.463} C_VEL
LIN {X 0,Y 607.916,Z 256.622,A -85,B 0,C 180,E1 29105.144,E2 29105.144} C_VEL
LIN {X 0,Y 607.904,Z 302.253,A -85,B 0,C 180,E1 29102.375,E2 29102.375} C_VEL
LIN {X 0,Y 607.911,Z 521.214,A -85,B 0,C 180,E1 29099.416,E2 29099.416} C_VEL
LIN {X 0,Y 607.904,Z 607.713,A -85,B 0,C 180,E1 29098.247,E2 29098.247} C_VEL
LIN {X 0,Y 607.906,Z 628.244,A -85,B 0,C 180,E1 29097.805,E2 29097.805} C_VEL
LIN {X 0,Y 607.906,Z 648.825,A -85,B 0,C 180,E1 29097.208,E2 29097.208} C_VEL
LIN {X 0,Y 607.913,Z 669.59,A -85,B 0,C 180,E1 29096.416,E2 29096.416} C_VEL
LIN {X 0,Y 607.918,Z 690.756,A -85,B 0,C 180,E1 29095.421,E2 29095.421} C_VEL
LIN {X 0,Y 607.916,Z 710.101,A -85,B 0,C 180,E1 29094.331,E2 29094.331} C_VEL
LIN {X 0,Y 607.914,Z 728.569,A -85,B 0,C 180,E1 29093.095,E2 29093.095} C_VEL
LIN {X 0,Y 607.911,Z 746.773,A -85,B 0,C 180,E1 29091.678,E2 29091.678} C_VEL
LIN {X 0,Y 607.913,Z 763.656,A -85,B 0,C 180,E1 29090.155,E2 29090.155} C_VEL
LIN {X 0,Y 607.918,Z 779.468,A -85,B 0,C 180,E1 29088.507,E2 29088.507} C_VEL
LIN {X 0,Y 607.913,Z 793.411,A -85,B 0,C 180,E1 29086.817,E2 29086.817} C_VEL
LIN {X 0,Y 607.918,Z 805.904,A -85,B 0,C 180,E1 29085.062,E2 29085.062} C_VEL
LIN {X 0,Y 607.919,Z 817.42,A -85,B 0,C 180,E1 29083.176,E2 29083.176} C_VEL
LIN {X 0,Y 607.912,Z 827.062,A -85,B 0,C 180,E1 29081.287,E2 29081.287} C_VEL
LIN {X 0,Y 607.911,Z 835.464,A -85,B 0,C 180,E1 29079.275,E2 29079.275} C_VEL
LIN {X 0,Y 607.91,Z 842.128,A -85,B 0,C 180,E1 29077.276,E2 29077.276} C_VEL
LIN {X 0,Y 607.912,Z 847.015,A -85,B 0,C 180,E1 29075.285,E2 29075.285} C_VEL
LIN {X 0,Y 607.917,Z 850.446,A -85,B 0,C 180,E1 29073.206,E2 29073.206} C_VEL
LIN {X 0,Y 607.91,Z 852.21,A -85,B 0,C 180,E1 29071.225,E2 29071.225} C_VEL
LIN {X 0,Y 607.902,Z 852.329,A -85,B 0,C 180,E1 29069.246,E2 29069.246} C_VEL
LIN {X 0,Y 607.908,Z 850.895,A -85,B 0,C 180,E1 29067.172,E2 29067.172} C_VEL
LIN {X 0,Y 607.912,Z 847.987,A -85,B 0,C 180,E1 29065.188,E2 29065.188} C_VEL
LIN {X 0,Y 607.915,Z 843.398,A -85,B 0,C 180,E1 29063.199,E2 29063.199} C_VEL
LIN {X 0,Y 607.906,Z 837.238,A -85,B 0,C 180,E1 29061.202,E2 29061.202} C_VEL
LIN {X 0,Y 607.899,Z 829.657,A -85,B 0,C 180,E1 29059.289,E2 29059.289} C_VEL
LIN {X 0,Y 607.899,Z 820.328,A -85,B 0,C 180,E1 29057.364,E2 29057.364} C_VEL
LIN {X 0,Y 607.904,Z 809.747,A -85,B 0,C 180,E1 29055.523,E2 29055.523} C_VEL
LIN {X 0,Y 607.911,Z 797.743,A -85,B 0,C 180,E1 29053.764,E2 29053.764} C_VEL
LIN {X 0,Y 607.906,Z 783.719,A -85,B 0,C 180,E1 29051.989,E2 29051.989} C_VEL
LIN {X 0,Y 607.908,Z 768.719,A -85,B 0,C 180,E1 29050.346,E2 29050.346} C_VEL
LIN {X 0,Y 607.916,Z 751.704,A -85,B 0,C 180,E1 29048.737,E2 29048.737} C_VEL
LIN {X 0,Y 607.918,Z 734.232,A -85,B 0,C 180,E1 29047.322,E2 29047.322} C_VEL
LIN {X 0,Y 607.915,Z 715.744,A -85,B 0,C 180,E1 29046.031,E2 29046.031} C_VEL
LIN {X 0,Y 607.918,Z 696.72,A -85,B 0,C 180,E1 29044.892,E2 29044.892} C_VEL
LIN {X 0,Y 607.901,Z 676.884,A -85,B 0,C 180,E1 29043.902,E2 29043.902} C_VEL
LIN {X 0,Y 607.906,Z 656.199,A -85,B 0,C 180,E1 29043.057,E2 29043.057} C_VEL
LIN {X 0,Y 607.917,Z 636.212,A -85,B 0,C 180,E1 29042.402,E2 29042.402} C_VEL
LIN {X 0,Y 607.903,Z 615.974,A -85,B 0,C 180,E1 29041.914,E2 29041.914} C_VEL
LIN {X 0,Y 607.913,Z 594.501,A -85,B 0,C 180,E1 29041.553,E2 29041.553} C_VEL
LIN {X 0,Y 607.908,Z 368.533,A -85,B 0,C 180,E1 29038.534,E2 29038.534} C_VEL
LIN {X 0,Y 607.906,Z 301.822,A -85,B 0,C 180,E1 29037.604,E2 29037.604} C_VEL
LIN {X 0,Y 607.91,Z 254.76,A -85,B 0,C 180,E1 29034.74,E2 29034.74} C_VEL
LIN {X 0,Y 607.897,Z 252.239,A -85,B 0,C 180,E1 29034.537,E2 29034.537} C_VEL
LIN {X 0,Y 607.881,Z 252.008,A -85,B 0,C 180,E1 29031.798,E2 29031.798} C_VEL
LIN {X 0,Y 607.901,Z 252.014,A -85,B 0,C 180,E1 29028.591,E2 29028.591} C_VEL
LIN {X 0,Y 607.903,Z 252.006,A -85,B 0,C 180,E1 29025.389,E2 29025.389} C_VEL
LIN {X 0,Y 607.867,Z 252.011,A -85,B 0,C 180,E1 29022.152,E2 29022.152} C_VEL
LIN {X 0,Y 607.917,Z 252.009,A -85,B 0,C 180,E1 29019.045,E2 29019.045} C_VEL
LIN {X 0,Y 607.856,Z 252.011,A -85,B 0,C 180,E1 29015.96,E2 29015.96} C_VEL
LIN {X 0,Y 607.918,Z 252.014,A -85,B 0,C 180,E1 29012.814,E2 29012.814} C_VEL
LIN {X 0,Y 607.849,Z 252.012,A -85,B 0,C 180,E1 29009.786,E2 29009.786} C_VEL
LIN {X 0,Y 607.91,Z 252.015,A -85,B 0,C 180,E1 29006.68,E2 29006.68} C_VEL
LIN {X 0,Y 607.84,Z 252.013,A -85,B 0,C 180,E1 29003.766,E2 29003.766} C_VEL
LIN {X 0,Y 607.91,Z 252.015,A -85,B 0,C 180,E1 29000.709,E2 29000.709} C_VEL
LIN {X 0,Y 607.83,Z 252.014,A -85,B 0,C 180,E1 28997.717,E2 28997.717} C_VEL
LIN {X 0,Y 607.903,Z 252.016,A -85,B 0,C 180,E1 28994.672,E2 28994.672} C_VEL
LIN {X 0,Y 607.829,Z 252.014,A -85,B 0,C 180,E1 28991.769,E2 28991.769} C_VEL
LIN {X 0,Y 607.907,Z 252.015,A -85,B 0,C 180,E1 28988.798,E2 28988.798} C_VEL
LIN {X 0,Y 607.838,Z 252.014,A -85,B 0,C 180,E1 28985.759,E2 28985.759} C_VEL
LIN {X 0,Y 607.903,Z 252.015,A -85,B 0,C 180,E1 28982.828,E2 28982.828} C_VEL
LIN {X 0,Y 607.846,Z 252.012,A -85,B 0,C 180,E1 28979.717,E2 28979.717} C_VEL
LIN {X 0,Y 607.917,Z 252.014,A -85,B 0,C 180,E1 28976.68,E2 28976.68} C_VEL
LIN {X 0,Y 606.914,Z 252.132,A -85,B 0,C 180,E1 28975.954,E2 28975.954} C_VEL
LIN {X 0,Y 600.441,Z 252.935,A -85,B 0,C 180,E1 28973.918,E2 28973.918} C_VEL
LIN {X 0,Y 599.918,Z 253.001,A -85,B 0,C 180,E1 28973.387,E2 28973.387} C_VEL
LIN {X 0,Y 599.962,Z 252.996,A -85,B 0,C 180,E1 28970.213,E2 28970.213} C_VEL
LIN {X 0,Y 599.933,Z 253.002,A -85,B 0,C 180,E1 28967.147,E2 28967.147} C_VEL
LIN {X 0,Y 599.94,Z 252.998,A -85,B 0,C 180,E1 28963.84,E2 28963.84} C_VEL
LIN {X 0,Y 599.97,Z 253.004,A -85,B 0,C 180,E1 28960.733,E2 28960.733} C_VEL
LIN {X 0,Y 599.936,Z 252.998,A -85,B 0,C 180,E1 28957.564,E2 28957.564} C_VEL
LIN {X 0,Y 599.972,Z 252.999,A -85,B 0,C 180,E1 28954.429,E2 28954.429} C_VEL
LIN {X 0,Y 599.942,Z 253,A -85,B 0,C 180,E1 28951.235,E2 28951.235} C_VEL
LIN {X 0,Y 599.978,Z 252.992,A -85,B 0,C 180,E1 28948.019,E2 28948.019} C_VEL
LIN {X 0,Y 599.974,Z 253.003,A -85,B 0,C 180,E1 28944.67,E2 28944.67} C_VEL
LIN {X 0,Y 599.952,Z 252.996,A -85,B 0,C 180,E1 28941.407,E2 28941.407} C_VEL
LIN {X 0,Y 599.962,Z 252.995,A -85,B 0,C 180,E1 28938.193,E2 28938.193} C_VEL
LIN {X 0,Y 599.959,Z 253.001,A -85,B 0,C 180,E1 28935.04,E2 28935.04} C_VEL
LIN {X 0,Y 599.969,Z 252.995,A -85,B 0,C 180,E1 28931.804,E2 28931.804} C_VEL
LIN {X 0,Y 599.968,Z 253.004,A -85,B 0,C 180,E1 28928.555,E2 28928.555} C_VEL
LIN {X 0,Y 599.966,Z 252.998,A -85,B 0,C 180,E1 28925.329,E2 28925.329} C_VEL
LIN {X 0,Y 599.992,Z 253.171,A -85,B 0,C 180,E1 28923.304,E2 28923.304} C_VEL
LIN {X 0,Y 600.818,Z 256.578,A -85,B 0,C 180,E1 28922.968,E2 28922.968} C_VEL
LIN {X 0,Y 600.66,Z 301.69,A -85,B 0,C 180,E1 28919.848,E2 28919.848} C_VEL
LIN {X 0,Y 600.672,Z 329.496,A -85,B 0,C 180,E1 28917.997,E2 28917.997} C_VEL
LIN {X 0,Y 600.686,Z 510.88,A -85,B 0,C 180,E1 28915.612,E2 28915.612} C_VEL
LIN {X 0,Y 600.611,Z 591.461,A -85,B 0,C 180,E1 28914.544,E2 28914.544} C_VEL
LIN {X 0,Y 600.558,Z 611.956,A -85,B 0,C 180,E1 28914.086,E2 28914.086} C_VEL
LIN {X 0,Y 600.498,Z 631.769,A -85,B 0,C 180,E1 28913.465,E2 28913.465} C_VEL
LIN {X 0,Y 600.428,Z 651.267,A -85,B 0,C 180,E1 28912.674,E2 28912.674} C_VEL
LIN {X 0,Y 600.347,Z 669.875,A -85,B 0,C 180,E1 28911.739,E2 28911.739} C_VEL
LIN {X 0,Y 600.277,Z 688.127,A -85,B 0,C 180,E1 28910.627,E2 28910.627} C_VEL
LIN {X 0,Y 600.195,Z 706.328,A -85,B 0,C 180,E1 28909.295,E2 28909.295} C_VEL
LIN {X 0,Y 600.124,Z 722.927,A -85,B 0,C 180,E1 28907.852,E2 28907.852} C_VEL
LIN {X 0,Y 600.06,Z 738.457,A -85,B 0,C 180,E1 28906.256,E2 28906.256} C_VEL
LIN {X 0,Y 600.008,Z 752.285,A -85,B 0,C 180,E1 28904.573,E2 28904.573} C_VEL
LIN {X 0,Y 599.97,Z 764.139,A -85,B 0,C 180,E1 28902.861,E2 28902.861} C_VEL
LIN {X 0,Y 599.939,Z 774.623,A -85,B 0,C 180,E1 28901.049,E2 28901.049} C_VEL
LIN {X 0,Y 599.932,Z 783.372,A -85,B 0,C 180,E1 28899.206,E2 28899.206} C_VEL
LIN {X 0,Y 599.912,Z 790.35,A -85,B 0,C 180,E1 28897.373,E2 28897.373} C_VEL
LIN {X 0,Y 599.906,Z 795.89,A -85,B 0,C 180,E1 28895.451,E2 28895.451} C_VEL
LIN {X 0,Y 599.903,Z 799.666,A -85,B 0,C 180,E1 28893.535,E2 28893.535} C_VEL
LIN {X 0,Y 599.904,Z 801.841,A -85,B 0,C 180,E1 28891.624,E2 28891.624} C_VEL
LIN {X 0,Y 599.904,Z 802.45,A -85,B 0,C 180,E1 28889.714,E2 28889.714} C_VEL
LIN {X 0,Y 599.909,Z 801.497,A -85,B 0,C 180,E1 28887.803,E2 28887.803} C_VEL
LIN {X 0,Y 599.912,Z 798.709,A -85,B 0,C 180,E1 28885.795,E2 28885.795} C_VEL
LIN {X 0,Y 599.919,Z 794.354,A -85,B 0,C 180,E1 28883.877,E2 28883.877} C_VEL
LIN {X 0,Y 599.928,Z 788.03,A -85,B 0,C 180,E1 28881.883,E2 28881.883} C_VEL
LIN {X 0,Y 599.93,Z 780.353,A -85,B 0,C 180,E1 28880.019,E2 28880.019} C_VEL
LIN {X 0,Y 599.943,Z 771.471,A -85,B 0,C 180,E1 28878.269,E2 28878.269} C_VEL
LIN {X 0,Y 599.972,Z 760.611,A -85,B 0,C 180,E1 28876.508,E2 28876.508} C_VEL
LIN {X 0,Y 600.017,Z 748.341,A -85,B 0,C 180,E1 28874.834,E2 28874.834} C_VEL
LIN {X 0,Y 600.065,Z 734.664,A -85,B 0,C 180,E1 28873.247,E2 28873.247} C_VEL
LIN {X 0,Y 600.132,Z 718.95,A -85,B 0,C 180,E1 28871.697,E2 28871.697} C_VEL
LIN {X 0,Y 600.206,Z 702.702,A -85,B 0,C 180,E1 28870.337,E2 28870.337} C_VEL
LIN {X 0,Y 600.289,Z 685.569,A -85,B 0,C 180,E1 28869.119,E2 28869.119} C_VEL
LIN {X 0,Y 600.372,Z 667.631,A -85,B 0,C 180,E1 28868.046,E2 28868.046} C_VEL
LIN {X 0,Y 600.435,Z 648.738,A -85,B 0,C 180,E1 28867.119,E2 28867.119} C_VEL
LIN {X 0,Y 600.504,Z 629.63,A -85,B 0,C 180,E1 28866.369,E2 28866.369} C_VEL
LIN {X 0,Y 600.563,Z 608.964,A -85,B 0,C 180,E1 28865.748,E2 28865.748} C_VEL
LIN {X 0,Y 600.615,Z 588.893,A -85,B 0,C 180,E1 28865.326,E2 28865.326} C_VEL
LIN {X 0,Y 600.818,Z 330.434,A -85,B 0,C 180,E1 28861.936,E2 28861.936} C_VEL
LIN {X 0,Y 600.58,Z 328.005,A -85,B 0,C 180,E1 28861.838,E2 28861.838} C_VEL
LIN {X 0,Y 600.731,Z 282.045,A -85,B 0,C 180,E1 28858.716,E2 28858.716} C_VEL
LIN {X 0,Y 600.677,Z 255.439,A -85,B 0,C 180,E1 28856.853,E2 28856.853} C_VEL
LIN {X 0,Y 599.999,Z 253.189,A -85,B 0,C 180,E1 28856.604,E2 28856.604} C_VEL
LIN {X 0,Y 599.966,Z 253,A -85,B 0,C 180,E1 28853.373,E2 28853.373} C_VEL
LIN {X 0,Y 599.959,Z 252.993,A -85,B 0,C 180,E1 28850.051,E2 28850.051} C_VEL
LIN {X 0,Y 599.962,Z 252.998,A -85,B 0,C 180,E1 28846.882,E2 28846.882} C_VEL
LIN {X 0,Y 599.958,Z 252.998,A -85,B 0,C 180,E1 28843.759,E2 28843.759} C_VEL
LIN {X 0,Y 599.956,Z 252.998,A -85,B 0,C 180,E1 28840.664,E2 28840.664} C_VEL
LIN {X 0,Y 599.967,Z 253,A -85,B 0,C 180,E1 28837.466,E2 28837.466} C_VEL
LIN {X 0,Y 599.965,Z 252.995,A -85,B 0,C 180,E1 28834.252,E2 28834.252} C_VEL
LIN {X 0,Y 599.96,Z 253,A -85,B 0,C 180,E1 28830.995,E2 28830.995} C_VEL
LIN {X 0,Y 599.971,Z 252.996,A -85,B 0,C 180,E1 28827.762,E2 28827.762} C_VEL
LIN {X 0,Y 599.941,Z 252.999,A -85,B 0,C 180,E1 28824.623,E2 28824.623} C_VEL
LIN {X 0,Y 599.972,Z 252.999,A -85,B 0,C 180,E1 28821.508,E2 28821.508} C_VEL
LIN {X 0,Y 599.936,Z 252.998,A -85,B 0,C 180,E1 28818.36,E2 28818.36} C_VEL
LIN {X 0,Y 599.968,Z 253.003,A -85,B 0,C 180,E1 28815.168,E2 28815.168} C_VEL
LIN {X 0,Y 599.943,Z 252.998,A -85,B 0,C 180,E1 28812.024,E2 28812.024} C_VEL
LIN {X 0,Y 599.93,Z 253.002,A -85,B 0,C 180,E1 28808.723,E2 28808.723} C_VEL
LIN {X 0,Y 599.971,Z 252.997,A -85,B 0,C 180,E1 28805.643,E2 28805.643} C_VEL
LIN {X 0,Y 599.915,Z 253.001,A -85,B 0,C 180,E1 28802.484,E2 28802.484} C_VEL
LIN {X 0,Y 599.979,Z 253.002,A -85,B 0,C 180,E1 28799.332,E2 28799.332} C_VEL
LIN {X 0,Y 599.906,Z 253.001,A -85,B 0,C 180,E1 28796.273,E2 28796.273} C_VEL
LIN {X 0,Y 599.969,Z 253.004,A -85,B 0,C 180,E1 28793.205,E2 28793.205} C_VEL
LIN {X 0,Y 599.896,Z 253.003,A -85,B 0,C 180,E1 28790.212,E2 28790.212} C_VEL
LIN {X 0,Y 599.956,Z 253.004,A -85,B 0,C 180,E1 28787.096,E2 28787.096} C_VEL
LIN {X 0,Y 599.889,Z 253.003,A -85,B 0,C 180,E1 28784.087,E2 28784.087} C_VEL
LIN {X 0,Y 599.956,Z 253.002,A -85,B 0,C 180,E1 28781.036,E2 28781.036} C_VEL
LIN {X 0,Y 599.898,Z 253.003,A -85,B 0,C 180,E1 28778.078,E2 28778.078} C_VEL
LIN {X 0,Y 599.959,Z 253.001,A -85,B 0,C 180,E1 28774.957,E2 28774.957} C_VEL
LIN {X 0,Y 599.909,Z 253.002,A -85,B 0,C 180,E1 28771.966,E2 28771.966} C_VEL
LIN {X 0,Y 599.948,Z 252.997,A -85,B 0,C 180,E1 28768.752,E2 28768.752} C_VEL
LIN {X 0,Y 599.924,Z 253.003,A -85,B 0,C 180,E1 28765.754,E2 28765.754} C_VEL
LIN {X 0,Y 599.931,Z 252.998,A -85,B 0,C 180,E1 28762.412,E2 28762.412} C_VEL
LIN {X 0,Y 599.972,Z 253.003,A -85,B 0,C 180,E1 28759.309,E2 28759.309} C_VEL
LIN {X 0,Y 599.928,Z 253,A -85,B 0,C 180,E1 28756.107,E2 28756.107} C_VEL
LIN {X 0,Y 599.975,Z 253,A -85,B 0,C 180,E1 28752.967,E2 28752.967} C_VEL
LIN {X 0,Y 599.937,Z 253.001,A -85,B 0,C 180,E1 28749.789,E2 28749.789} C_VEL
LIN {X 0,Y 599.966,Z 252.975,A -85,B 0,C 180,E1 28746.508,E2 28746.508} C_VEL
LIN {X 0,Y 599.994,Z 253.365,A -85,B 0,C 180,E1 28745.914,E2 28745.914} C_VEL
LIN {X 0,Y 601.027,Z 256.622,A -85,B 0,C 180,E1 28745.608,E2 28745.608} C_VEL
LIN {X 0,Y 600.97,Z 302.722,A -85,B 0,C 180,E1 28742.785,E2 28742.785} C_VEL
LIN {X 0,Y 600.994,Z 460.68,A -85,B 0,C 180,E1 28740.608,E2 28740.608} C_VEL
LIN {X 0,Y 600.847,Z 607.927,A -85,B 0,C 180,E1 28738.605,E2 28738.605} C_VEL
LIN {X 0,Y 600.787,Z 628.934,A -85,B 0,C 180,E1 28738.146,E2 28738.146} C_VEL
LIN {X 0,Y 600.711,Z 649.565,A -85,B 0,C 180,E1 28737.535,E2 28737.535} C_VEL
LIN {X 0,Y 600.646,Z 669.593,A -85,B 0,C 180,E1 28736.761,E2 28736.761} C_VEL
LIN {X 0,Y 600.54,Z 690.759,A -85,B 0,C 180,E1 28735.756,E2 28735.756} C_VEL
LIN {X 0,Y 600.444,Z 710.118,A -85,B 0,C 180,E1 28734.653,E2 28734.653} C_VEL
LIN {X 0,Y 600.354,Z 728.42,A -85,B 0,C 180,E1 28733.414,E2 28733.414} C_VEL
LIN {X 0,Y 600.249,Z 746.279,A -85,B 0,C 180,E1 28732.011,E2 28732.011} C_VEL
LIN {X 0,Y 600.166,Z 763.149,A -85,B 0,C 180,E1 28730.478,E2 28730.478} C_VEL
LIN {X 0,Y 600.103,Z 778.665,A -85,B 0,C 180,E1 28728.85,E2 28728.85} C_VEL
LIN {X 0,Y 600.048,Z 792.563,A -85,B 0,C 180,E1 28727.153,E2 28727.153} C_VEL
LIN {X 0,Y 599.999,Z 805.905,A -85,B 0,C 180,E1 28725.265,E2 28725.265} C_VEL
LIN {X 0,Y 599.958,Z 817.213,A -85,B 0,C 180,E1 28723.394,E2 28723.394} C_VEL
LIN {X 0,Y 599.931,Z 826.835,A -85,B 0,C 180,E1 28721.487,E2 28721.487} C_VEL
LIN {X 0,Y 599.915,Z 835.11,A -85,B 0,C 180,E1 28719.497,E2 28719.497} C_VEL
LIN {X 0,Y 599.912,Z 841.872,A -85,B 0,C 180,E1 28717.469,E2 28717.469} C_VEL
LIN {X 0,Y 599.915,Z 846.809,A -85,B 0,C 180,E1 28715.451,E2 28715.451} C_VEL
LIN {X 0,Y 599.916,Z 850.369,A -85,B 0,C 180,E1 28713.314,E2 28713.314} C_VEL
LIN {X 0,Y 599.909,Z 852.21,A -85,B 0,C 180,E1 28711.241,E2 28711.241} C_VEL
LIN {X 0,Y 599.903,Z 852.329,A -85,B 0,C 180,E1 28709.236,E2 28709.236} C_VEL
LIN {X 0,Y 599.909,Z 850.895,A -85,B 0,C 180,E1 28707.134,E2 28707.134} C_VEL
LIN {X 0,Y 599.913,Z 847.987,A -85,B 0,C 180,E1 28705.124,E2 28705.124} C_VEL
LIN {X 0,Y 599.921,Z 843.398,A -85,B 0,C 180,E1 28703.108,E2 28703.108} C_VEL
LIN {X 0,Y 599.924,Z 837.239,A -85,B 0,C 180,E1 28701.084,E2 28701.084} C_VEL
LIN {X 0,Y 599.923,Z 829.658,A -85,B 0,C 180,E1 28699.145,E2 28699.145} C_VEL
LIN {X 0,Y 599.943,Z 820.09,A -85,B 0,C 180,E1 28697.149,E2 28697.149} C_VEL
LIN {X 0,Y 599.978,Z 809.111,A -85,B 0,C 180,E1 28695.228,E2 28695.228} C_VEL
LIN {X 0,Y 600.013,Z 797.038,A -85,B 0,C 180,E1 28693.444,E2 28693.444} C_VEL
LIN {X 0,Y 600.082,Z 782.87,A -85,B 0,C 180,E1 28691.645,E2 28691.645} C_VEL
LIN {X 0,Y 600.155,Z 767.2,A -85,B 0,C 180,E1 28689.929,E2 28689.929} C_VEL
LIN {X 0,Y 600.242,Z 751.107,A -85,B 0,C 180,E1 28688.4,E2 28688.4} C_VEL
LIN {X 0,Y 600.312,Z 733.469,A -85,B 0,C 180,E1 28686.959,E2 28686.959} C_VEL
LIN {X 0,Y 600.418,Z 714.864,A -85,B 0,C 180,E1 28685.655,E2 28685.655} C_VEL
LIN {X 0,Y 600.529,Z 695.127,A -85,B 0,C 180,E1 28684.476,E2 28684.476} C_VEL
LIN {X 0,Y 600.594,Z 675.693,A -85,B 0,C 180,E1 28683.503,E2 28683.503} C_VEL
LIN {X 0,Y 600.692,Z 655.45,A -85,B 0,C 180,E1 28682.679,E2 28682.679} C_VEL
LIN {X 0,Y 600.788,Z 634.699,A -85,B 0,C 180,E1 28682.004,E2 28682.004} C_VEL
LIN {X 0,Y 600.824,Z 614.406,A -85,B 0,C 180,E1 28681.52,E2 28681.52} C_VEL
LIN {X 0,Y 600.886,Z 586.968,A -85,B 0,C 180,E1 28681.089,E2 28681.089} C_VEL
LIN {X 0,Y 601.079,Z 360.786,A -85,B 0,C 180,E1 28678.028,E2 28678.028} C_VEL
LIN {X 0,Y 600.964,Z 302.627,A -85,B 0,C 180,E1 28677.21,E2 28677.21} C_VEL
LIN {X 0,Y 601.029,Z 256.622,A -85,B 0,C 180,E1 28674.392,E2 28674.392} C_VEL
LIN {X 0,Y 599.969,Z 253.214,A -85,B 0,C 180,E1 28674.058,E2 28674.058} C_VEL
LIN {X 0,Y 599.973,Z 252.997,A -85,B 0,C 180,E1 28671.079,E2 28671.079} C_VEL
LIN {X 0,Y 599.933,Z 253,A -85,B 0,C 180,E1 28668.014,E2 28668.014} C_VEL
LIN {X 0,Y 599.976,Z 253,A -85,B 0,C 180,E1 28664.823,E2 28664.823} C_VEL
LIN {X 0,Y 599.932,Z 252.996,A -85,B 0,C 180,E1 28661.681,E2 28661.681} C_VEL
LIN {X 0,Y 599.943,Z 253.002,A -85,B 0,C 180,E1 28658.436,E2 28658.436} C_VEL
LIN {X 0,Y 599.94,Z 252.998,A -85,B 0,C 180,E1 28655.418,E2 28655.418} C_VEL
LIN {X 0,Y 599.919,Z 253,A -85,B 0,C 180,E1 28652.152,E2 28652.152} C_VEL
LIN {X 0,Y 599.96,Z 252.999,A -85,B 0,C 180,E1 28649.119,E2 28649.119} C_VEL
LIN {X 0,Y 599.906,Z 253.002,A -85,B 0,C 180,E1 28645.998,E2 28645.998} C_VEL
LIN {X 0,Y 599.969,Z 253.001,A -85,B 0,C 180,E1 28642.952,E2 28642.952} C_VEL
LIN {X 0,Y 599.897,Z 253.002,A -85,B 0,C 180,E1 28639.877,E2 28639.877} C_VEL
LIN {X 0,Y 599.965,Z 253.003,A -85,B 0,C 180,E1 28636.856,E2 28636.856} C_VEL
LIN {X 0,Y 599.889,Z 253.004,A -85,B 0,C 180,E1 28633.789,E2 28633.789} C_VEL
LIN {X 0,Y 599.958,Z 253.003,A -85,B 0,C 180,E1 28630.855,E2 28630.855} C_VEL
LIN {X 0,Y 599.896,Z 253.002,A -85,B 0,C 180,E1 28627.759,E2 28627.759} C_VEL
LIN {X 0,Y 599.975,Z 253.003,A -85,B 0,C 180,E1 28624.684,E2 28624.684} C_VEL
LIN {X 0,Y 599.904,Z 253.002,A -85,B 0,C 180,E1 28621.623,E2 28621.623} C_VEL
LIN {X 0,Y 599.98,Z 253,A -85,B 0,C 180,E1 28618.567,E2 28618.567} C_VEL
LIN {X 0,Y 599.913,Z 253.001,A -85,B 0,C 180,E1 28615.507,E2 28615.507} C_VEL
LIN {X 0,Y 599.918,Z 253.001,A -85,B 0,C 180,E1 28613.387,E2 28613.387} C_VEL
LIN {X 0,Y 598.961,Z 253.129,A -85,B 0,C 180,E1 28612.652,E2 28612.652} C_VEL
LIN {X 0,Y 592.474,Z 253.933,A -85,B 0,C 180,E1 28610.534,E2 28610.534} C_VEL
LIN {X 0,Y 592.007,Z 253.985,A -85,B 0,C 180,E1 28610.05,E2 28610.05} C_VEL
LIN {X 0,Y 592.014,Z 253.992,A -85,B 0,C 180,E1 28606.92,E2 28606.92} C_VEL
LIN {X 0,Y 591.995,Z 253.988,A -85,B 0,C 180,E1 28603.718,E2 28603.718} C_VEL
LIN {X 0,Y 592.038,Z 253.99,A -85,B 0,C 180,E1 28600.567,E2 28600.567} C_VEL
LIN {X 0,Y 591.996,Z 253.987,A -85,B 0,C 180,E1 28597.351,E2 28597.351} C_VEL
LIN {X 0,Y 592.035,Z 253.984,A -85,B 0,C 180,E1 28594.168,E2 28594.168} C_VEL
LIN {X 0,Y 592.022,Z 253.992,A -85,B 0,C 180,E1 28590.896,E2 28590.896} C_VEL
LIN {X 0,Y 592.012,Z 253.983,A -85,B 0,C 180,E1 28587.611,E2 28587.611} C_VEL
LIN {X 0,Y 592.031,Z 253.988,A -85,B 0,C 180,E1 28584.481,E2 28584.481} C_VEL
LIN {X 0,Y 592.012,Z 253.986,A -85,B 0,C 180,E1 28581.284,E2 28581.284} C_VEL
LIN {X 0,Y 592.028,Z 253.98,A -85,B 0,C 180,E1 28578.026,E2 28578.026} C_VEL
LIN {X 0,Y 592.035,Z 253.991,A -85,B 0,C 180,E1 28574.683,E2 28574.683} C_VEL
LIN {X 0,Y 592.024,Z 253.986,A -85,B 0,C 180,E1 28571.421,E2 28571.421} C_VEL
LIN {X 0,Y 592.016,Z 253.989,A -85,B 0,C 180,E1 28568.179,E2 28568.179} C_VEL
LIN {X 0,Y 592.027,Z 253.992,A -85,B 0,C 180,E1 28565.005,E2 28565.005} C_VEL
LIN {X 0,Y 592.063,Z 254.249,A -85,B 0,C 180,E1 28563.722,E2 28563.722} C_VEL
LIN {X 0,Y 593.729,Z 259.811,A -85,B 0,C 180,E1 28563.182,E2 28563.182} C_VEL
LIN {X 0,Y 593.414,Z 304.923,A -85,B 0,C 180,E1 28560.027,E2 28560.027} C_VEL
LIN {X 0,Y 593.364,Z 329.531,A -85,B 0,C 180,E1 28558.373,E2 28558.373} C_VEL
LIN {X 0,Y 593.757,Z 334.278,A -85,B 0,C 180,E1 28558.285,E2 28558.285} C_VEL
LIN {X 0,Y 593.335,Z 590.835,A -85,B 0,C 180,E1 28554.877,E2 28554.877} C_VEL
LIN {X 0,Y 593.231,Z 611.128,A -85,B 0,C 180,E1 28554.425,E2 28554.425} C_VEL
LIN {X 0,Y 593.107,Z 630.781,A -85,B 0,C 180,E1 28553.812,E2 28553.812} C_VEL
LIN {X 0,Y 592.956,Z 650.167,A -85,B 0,C 180,E1 28553.029,E2 28553.029} C_VEL
LIN {X 0,Y 592.819,Z 668.786,A -85,B 0,C 180,E1 28552.093,E2 28552.093} C_VEL
LIN {X 0,Y 592.663,Z 687.375,A -85,B 0,C 180,E1 28550.956,E2 28550.956} C_VEL
LIN {X 0,Y 592.498,Z 704.878,A -85,B 0,C 180,E1 28549.67,E2 28549.67} C_VEL
LIN {X 0,Y 592.349,Z 720.728,A -85,B 0,C 180,E1 28548.297,E2 28548.297} C_VEL
LIN {X 0,Y 592.219,Z 735.687,A -85,B 0,C 180,E1 28546.78,E2 28546.78} C_VEL
LIN {X 0,Y 592.123,Z 749.193,A -85,B 0,C 180,E1 28545.172,E2 28545.172} C_VEL
LIN {X 0,Y 592.038,Z 761.949,A -85,B 0,C 180,E1 28543.377,E2 28543.377} C_VEL
LIN {X 0,Y 591.974,Z 772.619,A -85,B 0,C 180,E1 28541.583,E2 28541.583} C_VEL
LIN {X 0,Y 591.947,Z 781.749,A -85,B 0,C 180,E1 28539.724,E2 28539.724} C_VEL
LIN {X 0,Y 591.931,Z 789.372,A -85,B 0,C 180,E1 28537.766,E2 28537.766} C_VEL
LIN {X 0,Y 591.922,Z 794.879,A -85,B 0,C 180,E1 28535.914,E2 28535.914} C_VEL
LIN {X 0,Y 591.919,Z 799.194,A -85,B 0,C 180,E1 28533.874,E2 28533.874} C_VEL
LIN {X 0,Y 591.916,Z 801.642,A -85,B 0,C 180,E1 28531.936,E2 28531.936} C_VEL
LIN {X 0,Y 591.915,Z 802.494,A -85,B 0,C 180,E1 28529.903,E2 28529.903} C_VEL
LIN {X 0,Y 591.912,Z 801.57,A -85,B 0,C 180,E1 28527.87,E2 28527.87} C_VEL
LIN {X 0,Y 591.916,Z 799.025,A -85,B 0,C 180,E1 28525.932,E2 28525.932} C_VEL
LIN {X 0,Y 591.924,Z 794.86,A -85,B 0,C 180,E1 28523.989,E2 28523.989} C_VEL
LIN {X 0,Y 591.932,Z 788.99,A -85,B 0,C 180,E1 28522.039,E2 28522.039} C_VEL
LIN {X 0,Y 591.949,Z 781.714,A -85,B 0,C 180,E1 28520.178,E2 28520.178} C_VEL
LIN {X 0,Y 591.974,Z 772.508,A -85,B 0,C 180,E1 28518.306,E2 28518.306} C_VEL
LIN {X 0,Y 592.036,Z 761.888,A -85,B 0,C 180,E1 28516.523,E2 28516.523} C_VEL
LIN {X 0,Y 592.117,Z 749.889,A -85,B 0,C 180,E1 28514.827,E2 28514.827} C_VEL
LIN {X 0,Y 592.22,Z 736.259,A -85,B 0,C 180,E1 28513.193,E2 28513.193} C_VEL
LIN {X 0,Y 592.344,Z 721.706,A -85,B 0,C 180,E1 28511.702,E2 28511.702} C_VEL
LIN {X 0,Y 592.498,Z 705.34,A -85,B 0,C 180,E1 28510.276,E2 28510.276} C_VEL
LIN {X 0,Y 592.657,Z 687.938,A -85,B 0,C 180,E1 28508.992,E2 28508.992} C_VEL
LIN {X 0,Y 592.808,Z 669.438,A -85,B 0,C 180,E1 28507.855,E2 28507.855} C_VEL
LIN {X 0,Y 592.954,Z 650.971,A -85,B 0,C 180,E1 28506.919,E2 28506.919} C_VEL
LIN {X 0,Y 593.107,Z 631.085,A -85,B 0,C 180,E1 28506.109,E2 28506.109} C_VEL
LIN {X 0,Y 593.23,Z 611.019,A -85,B 0,C 180,E1 28505.482,E2 28505.482} C_VEL
LIN {X 0,Y 593.335,Z 590.749,A -85,B 0,C 180,E1 28505.032,E2 28505.032} C_VEL
LIN {X 0,Y 593.751,Z 331.675,A -85,B 0,C 180,E1 28501.589,E2 28501.589} C_VEL
LIN {X 0,Y 593.279,Z 328.898,A -85,B 0,C 180,E1 28501.515,E2 28501.515} C_VEL
LIN {X 0,Y 593.565,Z 282.841,A -85,B 0,C 180,E1 28498.352,E2 28498.352} C_VEL
LIN {X 0,Y 593.663,Z 258.843,A -85,B 0,C 180,E1 28496.655,E2 28496.655} C_VEL
LIN {X 0,Y 592.06,Z 254.265,A -85,B 0,C 180,E1 28496.189,E2 28496.189} C_VEL
LIN {X 0,Y 592.028,Z 253.991,A -85,B 0,C 180,E1 28494.827,E2 28494.827} C_VEL
LIN {X 0,Y 592.016,Z 253.991,A -85,B 0,C 180,E1 28491.596,E2 28491.596} C_VEL
LIN {X 0,Y 592.038,Z 253.983,A -85,B 0,C 180,E1 28488.286,E2 28488.286} C_VEL
LIN {X 0,Y 592.026,Z 253.991,A -85,B 0,C 180,E1 28484.958,E2 28484.958} C_VEL
LIN {X 0,Y 592.021,Z 253.982,A -85,B 0,C 180,E1 28481.715,E2 28481.715} C_VEL
LIN {X 0,Y 592.018,Z 253.984,A -85,B 0,C 180,E1 28478.551,E2 28478.551} C_VEL
LIN {X 0,Y 592.032,Z 253.991,A -85,B 0,C 180,E1 28475.281,E2 28475.281} C_VEL
LIN {X 0,Y 592.035,Z 253.981,A -85,B 0,C 180,E1 28471.912,E2 28471.912} C_VEL
LIN {X 0,Y 592.009,Z 253.989,A -85,B 0,C 180,E1 28468.773,E2 28468.773} C_VEL
LIN {X 0,Y 592.032,Z 253.986,A -85,B 0,C 180,E1 28465.601,E2 28465.601} C_VEL
LIN {X 0,Y 592.001,Z 253.986,A -85,B 0,C 180,E1 28462.439,E2 28462.439} C_VEL
LIN {X 0,Y 592.034,Z 253.992,A -85,B 0,C 180,E1 28459.228,E2 28459.228} C_VEL
LIN {X 0,Y 592.008,Z 253.986,A -85,B 0,C 180,E1 28456.06,E2 28456.06} C_VEL
LIN {X 0,Y 591.997,Z 253.991,A -85,B 0,C 180,E1 28452.783,E2 28452.783} C_VEL
LIN {X 0,Y 592.035,Z 253.985,A -85,B 0,C 180,E1 28449.625,E2 28449.625} C_VEL
LIN {X 0,Y 591.981,Z 253.989,A -85,B 0,C 180,E1 28446.498,E2 28446.498} C_VEL
LIN {X 0,Y 592.039,Z 253.99,A -85,B 0,C 180,E1 28443.389,E2 28443.389} C_VEL
LIN {X 0,Y 591.972,Z 253.99,A -85,B 0,C 180,E1 28440.291,E2 28440.291} C_VEL
LIN {X 0,Y 592.033,Z 253.991,A -85,B 0,C 180,E1 28437.193,E2 28437.193} C_VEL
LIN {X 0,Y 591.966,Z 253.991,A -85,B 0,C 180,E1 28434.166,E2 28434.166} C_VEL
LIN {X 0,Y 591.999,Z 253.993,A -85,B 0,C 180,E1 28430.963,E2 28430.963} C_VEL
LIN {X 0,Y 591.961,Z 253.991,A -85,B 0,C 180,E1 28428.009,E2 28428.009} C_VEL
LIN {X 0,Y 591.971,Z 253.992,A -85,B 0,C 180,E1 28424.723,E2 28424.723} C_VEL
LIN {X 0,Y 591.961,Z 253.993,A -85,B 0,C 180,E1 28421.894,E2 28421.894} C_VEL
LIN {X 0,Y 591.968,Z 253.992,A -85,B 0,C 180,E1 28418.534,E2 28418.534} C_VEL
LIN {X 0,Y 591.985,Z 253.992,A -85,B 0,C 180,E1 28415.662,E2 28415.662} C_VEL
LIN {X 0,Y 591.975,Z 253.991,A -85,B 0,C 180,E1 28412.433,E2 28412.433} C_VEL
LIN {X 0,Y 592.013,Z 253.991,A -85,B 0,C 180,E1 28409.445,E2 28409.445} C_VEL
LIN {X 0,Y 591.977,Z 253.99,A -85,B 0,C 180,E1 28406.242,E2 28406.242} C_VEL
LIN {X 0,Y 592.039,Z 253.987,A -85,B 0,C 180,E1 28403.163,E2 28403.163} C_VEL
LIN {X 0,Y 591.983,Z 253.99,A -85,B 0,C 180,E1 28400.066,E2 28400.066} C_VEL
LIN {X 0,Y 592.038,Z 253.989,A -85,B 0,C 180,E1 28396.977,E2 28396.977} C_VEL
LIN {X 0,Y 591.993,Z 253.987,A -85,B 0,C 180,E1 28393.825,E2 28393.825} C_VEL
LIN {X 0,Y 592.025,Z 253.986,A -85,B 0,C 180,E1 28390.537,E2 28390.537} C_VEL
LIN {X 0,Y 592.024,Z 253.964,A -85,B 0,C 180,E1 28387.301,E2 28387.301} C_VEL
LIN {X 0,Y 592.065,Z 254.274,A -85,B 0,C 180,E1 28386.422,E2 28386.422} C_VEL
LIN {X 0,Y 594.168,Z 260.346,A -85,B 0,C 180,E1 28385.845,E2 28385.845} C_VEL
LIN {X 0,Y 593.988,Z 302.852,A -85,B 0,C 180,E1 28383.218,E2 28383.218} C_VEL
LIN {X 0,Y 594.398,Z 307.3,A -85,B 0,C 180,E1 28383.127,E2 28383.127} C_VEL
LIN {X 0,Y 593.97,Z 530.502,A -85,B 0,C 180,E1 28380.05,E2 28380.05} C_VEL
LIN {X 0,Y 593.813,Z 608.783,A -85,B 0,C 180,E1 28378.962,E2 28378.962} C_VEL
LIN {X 0,Y 593.689,Z 629.765,A -85,B 0,C 180,E1 28378.491,E2 28378.491} C_VEL
LIN {X 0,Y 593.534,Z 650.449,A -85,B 0,C 180,E1 28377.864,E2 28377.864} C_VEL
LIN {X 0,Y 593.398,Z 669.596,A -85,B 0,C 180,E1 28377.115,E2 28377.115} C_VEL
LIN {X 0,Y 593.182,Z 690.762,A -85,B 0,C 180,E1 28376.099,E2 28376.099} C_VEL
LIN {X 0,Y 593.004,Z 710.114,A -85,B 0,C 180,E1 28374.983,E2 28374.983} C_VEL
LIN {X 0,Y 592.809,Z 728.646,A -85,B 0,C 180,E1 28373.714,E2 28373.714} C_VEL
LIN {X 0,Y 592.599,Z 746.884,A -85,B 0,C 180,E1 28372.258,E2 28372.258} C_VEL
LIN {X 0,Y 592.423,Z 764.161,A -85,B 0,C 180,E1 28370.654,E2 28370.654} C_VEL
LIN {X 0,Y 592.292,Z 779.47,A -85,B 0,C 180,E1 28369.014,E2 28369.014} C_VEL
LIN {X 0,Y 592.178,Z 794.115,A -85,B 0,C 180,E1 28367.186,E2 28367.186} C_VEL
LIN {X 0,Y 592.081,Z 806.603,A -85,B 0,C 180,E1 28365.365,E2 28365.365} C_VEL
LIN {X 0,Y 592.004,Z 818.253,A -85,B 0,C 180,E1 28363.378,E2 28363.378} C_VEL
LIN {X 0,Y 591.959,Z 827.526,A -85,B 0,C 180,E1 28361.496,E2 28361.496} C_VEL
LIN {X 0,Y 591.927,Z 835.465,A -85,B 0,C 180,E1 28359.528,E2 28359.528} C_VEL
LIN {X 0,Y 591.919,Z 841.872,A -85,B 0,C 180,E1 28357.571,E2 28357.571} C_VEL
LIN {X 0,Y 591.917,Z 846.809,A -85,B 0,C 180,E1 28355.525,E2 28355.525} C_VEL
LIN {X 0,Y 591.917,Z 850.398,A -85,B 0,C 180,E1 28353.335,E2 28353.335} C_VEL
LIN {X 0,Y 591.908,Z 852.21,A -85,B 0,C 180,E1 28351.258,E2 28351.258} C_VEL
LIN {X 0,Y 591.903,Z 852.329,A -85,B 0,C 180,E1 28349.226,E2 28349.226} C_VEL
LIN {X 0,Y 591.911,Z 850.895,A -85,B 0,C 180,E1 28347.095,E2 28347.095} C_VEL
LIN {X 0,Y 591.916,Z 847.986,A -85,B 0,C 180,E1 28345.058,E2 28345.058} C_VEL
LIN {X 0,Y 591.924,Z 843.398,A -85,B 0,C 180,E1 28343.015,E2 28343.015} C_VEL
LIN {X 0,Y 591.941,Z 837.239,A -85,B 0,C 180,E1 28340.962,E2 28340.962} C_VEL
LIN {X 0,Y 591.952,Z 829.658,A -85,B 0,C 180,E1 28338.997,E2 28338.997} C_VEL
LIN {X 0,Y 591.989,Z 820.33,A -85,B 0,C 180,E1 28337.019,E2 28337.019} C_VEL
LIN {X 0,Y 592.055,Z 809.745,A -85,B 0,C 180,E1 28335.126,E2 28335.126} C_VEL
LIN {X 0,Y 592.125,Z 797.746,A -85,B 0,C 180,E1 28333.318,E2 28333.318} C_VEL
LIN {X 0,Y 592.254,Z 783.721,A -85,B 0,C 180,E1 28331.496,E2 28331.496} C_VEL
LIN {X 0,Y 592.401,Z 768.504,A -85,B 0,C 180,E1 28329.787,E2 28329.787} C_VEL
LIN {X 0,Y 592.566,Z 752.268,A -85,B 0,C 180,E1 28328.21,E2 28328.21} C_VEL
LIN {X 0,Y 592.718,Z 734.793,A -85,B 0,C 180,E1 28326.751,E2 28326.751} C_VEL
LIN {X 0,Y 592.933,Z 715.749,A -85,B 0,C 180,E1 28325.386,E2 28325.386} C_VEL
LIN {X 0,Y 593.151,Z 696.726,A -85,B 0,C 180,E1 28324.222,E2 28324.222} C_VEL
LIN {X 0,Y 593.301,Z 676.817,A -85,B 0,C 180,E1 28323.206,E2 28323.206} C_VEL
LIN {X 0,Y 593.499,Z 655.525,A -85,B 0,C 180,E1 28322.322,E2 28322.322} C_VEL
LIN {X 0,Y 593.682,Z 634.571,A -85,B 0,C 180,E1 28321.635,E2 28321.635} C_VEL
LIN {X 0,Y 593.77,Z 614.103,A -85,B 0,C 180,E1 28321.144,E2 28321.144} C_VEL
LIN {X 0,Y 593.882,Z 586.445,A -85,B 0,C 180,E1 28320.708,E2 28320.708} C_VEL
LIN {X 0,Y 594.289,Z 360.271,A -85,B 0,C 180,E1 28317.611,E2 28317.611} C_VEL
LIN {X 0,Y 594.213,Z 304.102,A -85,B 0,C 180,E1 28316.816,E2 28316.816} C_VEL
LIN {X 0,Y 593.877,Z 301.307,A -85,B 0,C 180,E1 28316.712,E2 28316.712} C_VEL
LIN {X 0,Y 594.114,Z 259.609,A -85,B 0,C 180,E1 28314.104,E2 28314.104} C_VEL
LIN {X 0,Y 592.061,Z 254.256,A -85,B 0,C 180,E1 28313.577,E2 28313.577} C_VEL
LIN {X 0,Y 592.005,Z 253.975,A -85,B 0,C 180,E1 28312.383,E2 28312.383} C_VEL
LIN {X 0,Y 592.038,Z 253.985,A -85,B 0,C 180,E1 28309.189,E2 28309.189} C_VEL
LIN {X 0,Y 591.991,Z 253.986,A -85,B 0,C 180,E1 28306.013,E2 28306.013} C_VEL
LIN {X 0,Y 592.039,Z 253.992,A -85,B 0,C 180,E1 28302.867,E2 28302.867} C_VEL
LIN {X 0,Y 591.986,Z 253.989,A -85,B 0,C 180,E1 28299.783,E2 28299.783} C_VEL
LIN {X 0,Y 592.021,Z 253.99,A -85,B 0,C 180,E1 28296.596,E2 28296.596} C_VEL
LIN {X 0,Y 591.989,Z 253.989,A -85,B 0,C 180,E1 28293.525,E2 28293.525} C_VEL
LIN {X 0,Y 591.983,Z 253.99,A -85,B 0,C 180,E1 28290.22,E2 28290.22} C_VEL
LIN {X 0,Y 592.002,Z 253.99,A -85,B 0,C 180,E1 28287.239,E2 28287.239} C_VEL
LIN {X 0,Y 591.967,Z 253.991,A -85,B 0,C 180,E1 28284.02,E2 28284.02} C_VEL
LIN {X 0,Y 592.019,Z 253.991,A -85,B 0,C 180,E1 28280.98,E2 28280.98} C_VEL
LIN {X 0,Y 591.955,Z 253.993,A -85,B 0,C 180,E1 28277.903,E2 28277.903} C_VEL
LIN {X 0,Y 592.019,Z 253.991,A -85,B 0,C 180,E1 28274.875,E2 28274.875} C_VEL
LIN {X 0,Y 591.952,Z 253.991,A -85,B 0,C 180,E1 28271.793,E2 28271.793} C_VEL
LIN {X 0,Y 592.032,Z 253.993,A -85,B 0,C 180,E1 28268.742,E2 28268.742} C_VEL
LIN {X 0,Y 591.961,Z 253.992,A -85,B 0,C 180,E1 28265.719,E2 28265.719} C_VEL
LIN {X 0,Y 592.038,Z 253.991,A -85,B 0,C 180,E1 28262.613,E2 28262.613} C_VEL
LIN {X 0,Y 591.969,Z 253.991,A -85,B 0,C 180,E1 28259.516,E2 28259.516} C_VEL
LIN {X 0,Y 592.033,Z 253.988,A -85,B 0,C 180,E1 28256.417,E2 28256.417} C_VEL
LIN {X 0,Y 591.982,Z 253.989,A -85,B 0,C 180,E1 28253.307,E2 28253.307} C_VEL
LIN {X 0,Y 592.007,Z 253.985,A -85,B 0,C 180,E1 28250.05,E2 28250.05} C_VEL
LIN {X 0,Y 590.978,Z 254.114,A -85,B 0,C 180,E1 28249.305,E2 28249.305} C_VEL
LIN {X 0,Y 584.603,Z 254.924,A -85,B 0,C 180,E1 28247.213,E2 28247.213} C_VEL
LIN {X 0,Y 584.098,Z 254.979,A -85,B 0,C 180,E1 28246.669,E2 28246.669} C_VEL
LIN {X 0,Y 584.051,Z 254.978,A -85,B 0,C 180,E1 28243.467,E2 28243.467} C_VEL
LIN {X 0,Y 584.099,Z 254.975,A -85,B 0,C 180,E1 28240.292,E2 28240.292} C_VEL
LIN {X 0,Y 584.069,Z 254.978,A -85,B 0,C 180,E1 28237.068,E2 28237.068} C_VEL
LIN {X 0,Y 584.069,Z 254.973,A -85,B 0,C 180,E1 28233.68,E2 28233.68} C_VEL
LIN {X 0,Y 584.093,Z 254.974,A -85,B 0,C 180,E1 28230.462,E2 28230.462} C_VEL
LIN {X 0,Y 584.068,Z 254.974,A -85,B 0,C 180,E1 28227.251,E2 28227.251} C_VEL
LIN {X 0,Y 584.096,Z 254.97,A -85,B 0,C 180,E1 28224.045,E2 28224.045} C_VEL
LIN {X 0,Y 584.098,Z 254.981,A -85,B 0,C 180,E1 28220.688,E2 28220.688} C_VEL
LIN {X 0,Y 584.078,Z 254.969,A -85,B 0,C 180,E1 28217.398,E2 28217.398} C_VEL
LIN {X 0,Y 584.082,Z 254.972,A -85,B 0,C 180,E1 28214.171,E2 28214.171} C_VEL
LIN {X 0,Y 584.086,Z 254.98,A -85,B 0,C 180,E1 28210.966,E2 28210.966} C_VEL
LIN {X 0,Y 584.097,Z 254.974,A -85,B 0,C 180,E1 28207.669,E2 28207.669} C_VEL
LIN {X 0,Y 584.08,Z 254.971,A -85,B 0,C 180,E1 28204.395,E2 28204.395} C_VEL
LIN {X 0,Y 584.159,Z 255.51,A -85,B 0,C 180,E1 28204.13,E2 28204.13} C_VEL
LIN {X 0,Y 586.654,Z 262.238,A -85,B 0,C 180,E1 28203.459,E2 28203.459} C_VEL
LIN {X 0,Y 586.177,Z 307.351,A -85,B 0,C 180,E1 28200.267,E2 28200.267} C_VEL
LIN {X 0,Y 586.07,Z 329.57,A -85,B 0,C 180,E1 28198.759,E2 28198.759} C_VEL
LIN {X 0,Y 586.712,Z 334.722,A -85,B 0,C 180,E1 28198.651,E2 28198.651} C_VEL
LIN {X 0,Y 586.074,Z 590.667,A -85,B 0,C 180,E1 28195.21,E2 28195.21} C_VEL
LIN {X 0,Y 585.921,Z 610.87,A -85,B 0,C 180,E1 28194.757,E2 28194.757} C_VEL
LIN {X 0,Y 585.732,Z 630.803,A -85,B 0,C 180,E1 28194.131,E2 28194.131} C_VEL
LIN {X 0,Y 585.497,Z 650.88,A -85,B 0,C 180,E1 28193.306,E2 28193.306} C_VEL
LIN {X 0,Y 585.279,Z 669.695,A -85,B 0,C 180,E1 28192.34,E2 28192.34} C_VEL
LIN {X 0,Y 585.056,Z 687.387,A -85,B 0,C 180,E1 28191.241,E2 28191.241} C_VEL
LIN {X 0,Y 584.803,Z 704.852,A -85,B 0,C 180,E1 28189.943,E2 28189.943} C_VEL
LIN {X 0,Y 584.584,Z 720.736,A -85,B 0,C 180,E1 28188.549,E2 28188.549} C_VEL
LIN {X 0,Y 584.384,Z 735.693,A -85,B 0,C 180,E1 28187.012,E2 28187.012} C_VEL
LIN {X 0,Y 584.237,Z 749.2,A -85,B 0,C 180,E1 28185.382,E2 28185.382} C_VEL
LIN {X 0,Y 584.105,Z 761.954,A -85,B 0,C 180,E1 28183.563,E2 28183.563} C_VEL
LIN {X 0,Y 584.017,Z 772.56,A -85,B 0,C 180,E1 28181.755,E2 28181.755} C_VEL
LIN {X 0,Y 583.968,Z 781.752,A -85,B 0,C 180,E1 28179.858,E2 28179.858} C_VEL
LIN {X 0,Y 583.939,Z 789.374,A -85,B 0,C 180,E1 28177.873,E2 28177.873} C_VEL
LIN {X 0,Y 583.925,Z 794.881,A -85,B 0,C 180,E1 28175.995,E2 28175.995} C_VEL
LIN {X 0,Y 583.92,Z 799.196,A -85,B 0,C 180,E1 28173.927,E2 28173.927} C_VEL
LIN {X 0,Y 583.916,Z 801.642,A -85,B 0,C 180,E1 28171.963,E2 28171.963} C_VEL
LIN {X 0,Y 583.914,Z 802.493,A -85,B 0,C 180,E1 28169.902,E2 28169.902} C_VEL
LIN {X 0,Y 583.911,Z 801.569,A -85,B 0,C 180,E1 28167.841,E2 28167.841} C_VEL
LIN {X 0,Y 583.915,Z 799.024,A -85,B 0,C 180,E1 28165.876,E2 28165.876} C_VEL
LIN {X 0,Y 583.925,Z 794.859,A -85,B 0,C 180,E1 28163.906,E2 28163.906} C_VEL
LIN {X 0,Y 583.942,Z 788.988,A -85,B 0,C 180,E1 28161.929,E2 28161.929} C_VEL
LIN {X 0,Y 583.97,Z 781.712,A -85,B 0,C 180,E1 28160.042,E2 28160.042} C_VEL
LIN {X 0,Y 584.017,Z 772.506,A -85,B 0,C 180,E1 28158.145,E2 28158.145} C_VEL
LIN {X 0,Y 584.104,Z 761.885,A -85,B 0,C 180,E1 28156.337,E2 28156.337} C_VEL
LIN {X 0,Y 584.229,Z 749.885,A -85,B 0,C 180,E1 28154.617,E2 28154.617} C_VEL
LIN {X 0,Y 584.379,Z 736.506,A -85,B 0,C 180,E1 28152.988,E2 28152.988} C_VEL
LIN {X 0,Y 584.575,Z 721.701,A -85,B 0,C 180,E1 28151.45,E2 28151.45} C_VEL
LIN {X 0,Y 584.801,Z 705.335,A -85,B 0,C 180,E1 28150.005,E2 28150.005} C_VEL
LIN {X 0,Y 585.049,Z 687.852,A -85,B 0,C 180,E1 28148.701,E2 28148.701} C_VEL
LIN {X 0,Y 585.288,Z 669.318,A -85,B 0,C 180,E1 28147.549,E2 28147.549} C_VEL
LIN {X 0,Y 585.501,Z 650.961,A -85,B 0,C 180,E1 28146.607,E2 28146.607} C_VEL
LIN {X 0,Y 585.729,Z 630.997,A -85,B 0,C 180,E1 28145.786,E2 28145.786} C_VEL
LIN {X 0,Y 585.921,Z 610.865,A -85,B 0,C 180,E1 28145.152,E2 28145.152} C_VEL
LIN {X 0,Y 586.074,Z 590.58,A -85,B 0,C 180,E1 28144.699,E2 28144.699} C_VEL
LIN {X 0,Y 586.707,Z 333.001,A -85,B 0,C 180,E1 28141.236,E2 28141.236} C_VEL
LIN {X 0,Y 585.982,Z 328.897,A -85,B 0,C 180,E1 28141.127,E2 28141.127} C_VEL
LIN {X 0,Y 586.423,Z 283.637,A -85,B 0,C 180,E1 28137.978,E2 28137.978} C_VEL
LIN {X 0,Y 586.47,Z 261.574,A -85,B 0,C 180,E1 28136.391,E2 28136.391} C_VEL
LIN {X 0,Y 584.124,Z 255.337,A -85,B 0,C 180,E1 28135.753,E2 28135.753} C_VEL
LIN {X 0,Y 584.095,Z 254.977,A -85,B 0,C 180,E1 28135.129,E2 28135.129} C_VEL
LIN {X 0,Y 584.076,Z 254.978,A -85,B 0,C 180,E1 28131.949,E2 28131.949} C_VEL
LIN {X 0,Y 584.086,Z 254.977,A -85,B 0,C 180,E1 28128.72,E2 28128.72} C_VEL
LIN {X 0,Y 584.088,Z 254.976,A -85,B 0,C 180,E1 28125.426,E2 28125.426} C_VEL
LIN {X 0,Y 584.095,Z 254.965,A -85,B 0,C 180,E1 28122.147,E2 28122.147} C_VEL
LIN {X 0,Y 584.079,Z 254.976,A -85,B 0,C 180,E1 28118.843,E2 28118.843} C_VEL
LIN {X 0,Y 584.088,Z 254.974,A -85,B 0,C 180,E1 28115.593,E2 28115.593} C_VEL
LIN {X 0,Y 584.076,Z 254.971,A -85,B 0,C 180,E1 28112.399,E2 28112.399} C_VEL
LIN {X 0,Y 584.09,Z 254.981,A -85,B 0,C 180,E1 28109.089,E2 28109.089} C_VEL
LIN {X 0,Y 584.095,Z 254.972,A -85,B 0,C 180,E1 28105.773,E2 28105.773} C_VEL
LIN {X 0,Y 584.062,Z 254.975,A -85,B 0,C 180,E1 28102.549,E2 28102.549} C_VEL
LIN {X 0,Y 584.097,Z 254.981,A -85,B 0,C 180,E1 28099.292,E2 28099.292} C_VEL
LIN {X 0,Y 584.066,Z 254.976,A -85,B 0,C 180,E1 28096.101,E2 28096.101} C_VEL
LIN {X 0,Y 584.057,Z 254.98,A -85,B 0,C 180,E1 28092.758,E2 28092.758} C_VEL
LIN {X 0,Y 584.098,Z 254.974,A -85,B 0,C 180,E1 28089.558,E2 28089.558} C_VEL
LIN {X 0,Y 584.042,Z 254.977,A -85,B 0,C 180,E1 28086.389,E2 28086.389} C_VEL
LIN {X 0,Y 584.096,Z 254.982,A -85,B 0,C 180,E1 28083.239,E2 28083.239} C_VEL
LIN {X 0,Y 584.036,Z 254.979,A -85,B 0,C 180,E1 28080.196,E2 28080.196} C_VEL
LIN {X 0,Y 584.063,Z 254.981,A -85,B 0,C 180,E1 28076.958,E2 28076.958} C_VEL
LIN {X 0,Y 584.034,Z 254.98,A -85,B 0,C 180,E1 28074.006,E2 28074.006} C_VEL
LIN {X 0,Y 584.03,Z 254.982,A -85,B 0,C 180,E1 28070.64,E2 28070.64} C_VEL
LIN {X 0,Y 584.04,Z 254.979,A -85,B 0,C 180,E1 28067.744,E2 28067.744} C_VEL
LIN {X 0,Y 584.017,Z 254.98,A -85,B 0,C 180,E1 28064.51,E2 28064.51} C_VEL
LIN {X 0,Y 584.055,Z 254.982,A -85,B 0,C 180,E1 28061.536,E2 28061.536} C_VEL
LIN {X 0,Y 584.022,Z 254.981,A -85,B 0,C 180,E1 28058.373,E2 28058.373} C_VEL
LIN {X 0,Y 584.087,Z 254.982,A -85,B 0,C 180,E1 28055.312,E2 28055.312} C_VEL
LIN {X 0,Y 584.031,Z 254.98,A -85,B 0,C 180,E1 28052.247,E2 28052.247} C_VEL
LIN {X 0,Y 584.101,Z 254.972,A -85,B 0,C 180,E1 28049.101,E2 28049.101} C_VEL
LIN {X 0,Y 584.039,Z 254.98,A -85,B 0,C 180,E1 28045.952,E2 28045.952} C_VEL
LIN {X 0,Y 584.078,Z 254.974,A -85,B 0,C 180,E1 28042.7,E2 28042.7} C_VEL
LIN {X 0,Y 584.061,Z 254.981,A -85,B 0,C 180,E1 28039.621,E2 28039.621} C_VEL
LIN {X 0,Y 584.062,Z 254.977,A -85,B 0,C 180,E1 28036.378,E2 28036.378} C_VEL
LIN {X 0,Y 584.097,Z 254.98,A -85,B 0,C 180,E1 28033.179,E2 28033.179} C_VEL
LIN {X 0,Y 584.057,Z 254.979,A -85,B 0,C 180,E1 28029.92,E2 28029.92} C_VEL
LIN {X 0,Y 584.127,Z 255.193,A -85,B 0,C 180,E1 28026.954,E2 28026.954} C_VEL
LIN {X 0,Y 585.462,Z 258.591,A -85,B 0,C 180,E1 28026.578,E2 28026.578} C_VEL
LIN {X 0,Y 587.319,Z 263.138,A -85,B 0,C 180,E1 28026.148,E2 28026.148} C_VEL
LIN {X 0,Y 586.933,Z 302.216,A -85,B 0,C 180,E1 28023.686,E2 28023.686} C_VEL
LIN {X 0,Y 587.692,Z 308.121,A -85,B 0,C 180,E1 28023.543,E2 28023.543} C_VEL
LIN {X 0,Y 587.041,Z 531.138,A -85,B 0,C 180,E1 28020.433,E2 28020.433} C_VEL
LIN {X 0,Y 586.805,Z 608.997,A -85,B 0,C 180,E1 28019.338,E2 28019.338} C_VEL
LIN {X 0,Y 586.614,Z 630.025,A -85,B 0,C 180,E1 28018.86,E2 28018.86} C_VEL
LIN {X 0,Y 586.368,Z 651.778,A -85,B 0,C 180,E1 28018.185,E2 28018.185} C_VEL
LIN {X 0,Y 586.153,Z 672.145,A -85,B 0,C 180,E1 28017.368,E2 28017.368} C_VEL
LIN {X 0,Y 585.832,Z 692.456,A -85,B 0,C 180,E1 28016.359,E2 28016.359} C_VEL
LIN {X 0,Y 585.521,Z 712.541,A -85,B 0,C 180,E1 28015.163,E2 28015.163} C_VEL
LIN {X 0,Y 585.249,Z 731.462,A -85,B 0,C 180,E1 28013.831,E2 28013.831} C_VEL
LIN {X 0,Y 584.944,Z 749.1,A -85,B 0,C 180,E1 28012.371,E2 28012.371} C_VEL
LIN {X 0,Y 584.68,Z 765.68,A -85,B 0,C 180,E1 28010.783,E2 28010.783} C_VEL
LIN {X 0,Y 584.466,Z 781.171,A -85,B 0,C 180,E1 28009.071,E2 28009.071} C_VEL
LIN {X 0,Y 584.303,Z 795.627,A -85,B 0,C 180,E1 28007.219,E2 28007.219} C_VEL
LIN {X 0,Y 584.159,Z 808.473,A -85,B 0,C 180,E1 28005.283,E2 28005.283} C_VEL
LIN {X 0,Y 584.051,Z 819.292,A -85,B 0,C 180,E1 28003.362,E2 28003.362} C_VEL
LIN {X 0,Y 583.988,Z 828.844,A -85,B 0,C 180,E1 28001.355,E2 28001.355} C_VEL
LIN {X 0,Y 583.944,Z 836.53,A -85,B 0,C 180,E1 27999.361,E2 27999.361} C_VEL
LIN {X 0,Y 583.927,Z 843.145,A -85,B 0,C 180,E1 27997.18,E2 27997.18} C_VEL
LIN {X 0,Y 583.918,Z 847.825,A -85,B 0,C 180,E1 27995.108,E2 27995.108} C_VEL
LIN {X 0,Y 583.915,Z 850.784,A -85,B 0,C 180,E1 27993.043,E2 27993.043} C_VEL
LIN {X 0,Y 583.909,Z 852.306,A -85,B 0,C 180,E1 27990.883,E2 27990.883} C_VEL
LIN {X 0,Y 583.912,Z 852.239,A -85,B 0,C 180,E1 27988.823,E2 27988.823} C_VEL
LIN {X 0,Y 583.917,Z 850.559,A -85,B 0,C 180,E1 27986.761,E2 27986.761} C_VEL
LIN {X 0,Y 583.917,Z 847.22,A -85,B 0,C 180,E1 27984.596,E2 27984.596} C_VEL
LIN {X 0,Y 583.92,Z 842.636,A -85,B 0,C 180,E1 27982.622,E2 27982.622} C_VEL
LIN {X 0,Y 583.94,Z 836.003,A -85,B 0,C 180,E1 27980.491,E2 27980.491} C_VEL
LIN {X 0,Y 583.989,Z 828.432,A -85,B 0,C 180,E1 27978.545,E2 27978.545} C_VEL
LIN {X 0,Y 584.051,Z 818.773,A -85,B 0,C 180,E1 27976.537,E2 27976.537} C_VEL
LIN {X 0,Y 584.163,Z 807.104,A -85,B 0,C 180,E1 27974.5,E2 27974.5} C_VEL
LIN {X 0,Y 584.312,Z 794.884,A -85,B 0,C 180,E1 27972.678,E2 27972.678} C_VEL
LIN {X 0,Y 584.482,Z 780.321,A -85,B 0,C 180,E1 27970.826,E2 27970.826} C_VEL
LIN {X 0,Y 584.686,Z 765.174,A -85,B 0,C 180,E1 27969.164,E2 27969.164} C_VEL
LIN {X 0,Y 584.962,Z 747.489,A -85,B 0,C 180,E1 27967.489,E2 27967.489} C_VEL
LIN {X 0,Y 585.267,Z 730.004,A -85,B 0,C 180,E1 27966.061,E2 27966.061} C_VEL
LIN {X 0,Y 585.543,Z 711.735,A -85,B 0,C 180,E1 27964.784,E2 27964.784} C_VEL
LIN {X 0,Y 585.838,Z 691.761,A -85,B 0,C 180,E1 27963.603,E2 27963.603} C_VEL
LIN {X 0,Y 586.153,Z 672.145,A -85,B 0,C 180,E1 27962.632,E2 27962.632} C_VEL
LIN {X 0,Y 586.368,Z 651.781,A -85,B 0,C 180,E1 27961.815,E2 27961.815} C_VEL
LIN {X 0,Y 586.618,Z 629.901,A -85,B 0,C 180,E1 27961.137,E2 27961.137} C_VEL
LIN {X 0,Y 586.809,Z 608.785,A -85,B 0,C 180,E1 27960.658,E2 27960.658} C_VEL
LIN {X 0,Y 587.065,Z 524.14,A -85,B 0,C 180,E1 27959.471,E2 27959.471} C_VEL
LIN {X 0,Y 587.671,Z 306.443,A -85,B 0,C 180,E1 27956.431,E2 27956.431} C_VEL
LIN {X 0,Y 586.906,Z 301.307,A -85,B 0,C 180,E1 27956.264,E2 27956.264} C_VEL
LIN {X 0,Y 587.319,Z 263.138,A -85,B 0,C 180,E1 27953.852,E2 27953.852} C_VEL
LIN {X 0,Y 584.137,Z 255.259,A -85,B 0,C 180,E1 27953.068,E2 27953.068} C_VEL
LIN {X 0,Y 584.059,Z 254.962,A -85,B 0,C 180,E1 27952.08,E2 27952.08} C_VEL
LIN {X 0,Y 584.098,Z 254.972,A -85,B 0,C 180,E1 27948.867,E2 27948.867} C_VEL
LIN {X 0,Y 584.061,Z 254.972,A -85,B 0,C 180,E1 27945.69,E2 27945.69} C_VEL
LIN {X 0,Y 584.058,Z 254.975,A -85,B 0,C 180,E1 27942.309,E2 27942.309} C_VEL
LIN {X 0,Y 584.097,Z 254.976,A -85,B 0,C 180,E1 27939.157,E2 27939.157} C_VEL
LIN {X 0,Y 584.041,Z 254.977,A -85,B 0,C 180,E1 27935.959,E2 27935.959} C_VEL
LIN {X 0,Y 584.096,Z 254.978,A -85,B 0,C 180,E1 27932.747,E2 27932.747} C_VEL
LIN {X 0,Y 584.036,Z 254.977,A -85,B 0,C 180,E1 27929.654,E2 27929.654} C_VEL
LIN {X 0,Y 584.059,Z 254.981,A -85,B 0,C 180,E1 27926.429,E2 27926.429} C_VEL
LIN {X 0,Y 584.032,Z 254.979,A -85,B 0,C 180,E1 27923.509,E2 27923.509} C_VEL
LIN {X 0,Y 584.031,Z 254.98,A -85,B 0,C 180,E1 27920.127,E2 27920.127} C_VEL
LIN {X 0,Y 584.042,Z 254.981,A -85,B 0,C 180,E1 27917.206,E2 27917.206} C_VEL
LIN {X 0,Y 584.017,Z 254.982,A -85,B 0,C 180,E1 27913.969,E2 27913.969} C_VEL
LIN {X 0,Y 584.053,Z 254.98,A -85,B 0,C 180,E1 27911.054,E2 27911.054} C_VEL
LIN {X 0,Y 584.022,Z 254.98,A -85,B 0,C 180,E1 27907.872,E2 27907.872} C_VEL
LIN {X 0,Y 584.073,Z 254.982,A -85,B 0,C 180,E1 27904.91,E2 27904.91} C_VEL
LIN {X 0,Y 584.028,Z 254.98,A -85,B 0,C 180,E1 27901.766,E2 27901.766} C_VEL
LIN {X 0,Y 584.094,Z 254.98,A -85,B 0,C 180,E1 27898.725,E2 27898.725} C_VEL
LIN {X 0,Y 584.036,Z 254.979,A -85,B 0,C 180,E1 27895.581,E2 27895.581} C_VEL
LIN {X 0,Y 584.101,Z 254.977,A -85,B 0,C 180,E1 27892.426,E2 27892.426} C_VEL
LIN {X 0,Y 584.05,Z 254.977,A -85,B 0,C 180,E1 27889.245,E2 27889.245} C_VEL
LIN {X 0,Y 584.098,Z 254.979,A -85,B 0,C 180,E1 27886.669,E2 27886.669} C_VEL
LIN {X 0,Y 583.121,Z 255.094,A -85,B 0,C 180,E1 27885.913,E2 27885.913} C_VEL
LIN {X 0,Y 576.638,Z 255.902,A -85,B 0,C 180,E1 27883.793,E2 27883.793} C_VEL
LIN {X 0,Y 576.117,Z 255.968,A -85,B 0,C 180,E1 27883.24,E2 27883.24} C_VEL
LIN {X 0,Y 576.135,Z 255.964,A -85,B 0,C 180,E1 27879.902,E2 27879.902} C_VEL
LIN {X 0,Y 576.159,Z 255.969,A -85,B 0,C 180,E1 27876.634,E2 27876.634} C_VEL
LIN {X 0,Y 576.123,Z 255.964,A -85,B 0,C 180,E1 27873.349,E2 27873.349} C_VEL
LIN {X 0,Y 576.157,Z 255.958,A -85,B 0,C 180,E1 27870.128,E2 27870.128} C_VEL
LIN {X 0,Y 576.151,Z 255.967,A -85,B 0,C 180,E1 27866.766,E2 27866.766} C_VEL
LIN {X 0,Y 576.135,Z 255.96,A -85,B 0,C 180,E1 27863.465,E2 27863.465} C_VEL
LIN {X 0,Y 576.149,Z 255.966,A -85,B 0,C 180,E1 27860.243,E2 27860.243} C_VEL
LIN {X 0,Y 576.146,Z 255.96,A -85,B 0,C 180,E1 27856.936,E2 27856.936} C_VEL
LIN {X 0,Y 576.151,Z 255.957,A -85,B 0,C 180,E1 27853.546,E2 27853.546} C_VEL
LIN {X 0,Y 576.143,Z 255.961,A -85,B 0,C 180,E1 27850.338,E2 27850.338} C_VEL
LIN {X 0,Y 576.146,Z 255.966,A -85,B 0,C 180,E1 27847.151,E2 27847.151} C_VEL
LIN {X 0,Y 576.188,Z 256.191,A -85,B 0,C 180,E1 27844.645,E2 27844.645} C_VEL
LIN {X 0,Y 579.011,Z 263.897,A -85,B 0,C 180,E1 27843.838,E2 27843.838} C_VEL
LIN {X 0,Y 579.583,Z 265.391,A -85,B 0,C 180,E1 27843.69,E2 27843.69} C_VEL
LIN {X 0,Y 578.945,Z 310.221,A -85,B 0,C 180,E1 27840.481,E2 27840.481} C_VEL
LIN {X 0,Y 578.717,Z 329.038,A -85,B 0,C 180,E1 27839.174,E2 27839.174} C_VEL
LIN {X 0,Y 579.689,Z 335.837,A -85,B 0,C 180,E1 27839.016,E2 27839.016} C_VEL
LIN {X 0,Y 578.834,Z 590.497,A -85,B 0,C 180,E1 27835.551,E2 27835.551} C_VEL
LIN {X 0,Y 578.631,Z 610.8,A -85,B 0,C 180,E1 27835.093,E2 27835.093} C_VEL
LIN {X 0,Y 578.375,Z 630.824,A -85,B 0,C 180,E1 27834.458,E2 27834.458} C_VEL
LIN {X 0,Y 578.083,Z 650.195,A -85,B 0,C 180,E1 27833.657,E2 27833.657} C_VEL
LIN {X 0,Y 577.795,Z 668.804,A -85,B 0,C 180,E1 27832.699,E2 27832.699} C_VEL
LIN {X 0,Y 577.461,Z 687.398,A -85,B 0,C 180,E1 27831.535,E2 27831.535} C_VEL
LIN {X 0,Y 577.123,Z 704.64,A -85,B 0,C 180,E1 27830.238,E2 27830.238} C_VEL
LIN {X 0,Y 576.826,Z 720.744,A -85,B 0,C 180,E1 27828.808,E2 27828.808} C_VEL
LIN {X 0,Y 576.56,Z 735.699,A -85,B 0,C 180,E1 27827.25,E2 27827.25} C_VEL
LIN {X 0,Y 576.358,Z 749.206,A -85,B 0,C 180,E1 27825.598,E2 27825.598} C_VEL
LIN {X 0,Y 576.184,Z 761.959,A -85,B 0,C 180,E1 27823.753,E2 27823.753} C_VEL
LIN {X 0,Y 576.065,Z 772.564,A -85,B 0,C 180,E1 27821.92,E2 27821.92} C_VEL
LIN {X 0,Y 575.992,Z 781.755,A -85,B 0,C 180,E1 27819.996,E2 27819.996} C_VEL
LIN {X 0,Y 575.949,Z 789.376,A -85,B 0,C 180,E1 27817.983,E2 27817.983} C_VEL
LIN {X 0,Y 575.928,Z 794.883,A -85,B 0,C 180,E1 27816.079,E2 27816.079} C_VEL
LIN {X 0,Y 575.919,Z 799.197,A -85,B 0,C 180,E1 27813.982,E2 27813.982} C_VEL
LIN {X 0,Y 575.916,Z 801.642,A -85,B 0,C 180,E1 27811.99,E2 27811.99} C_VEL
LIN {X 0,Y 575.914,Z 802.493,A -85,B 0,C 180,E1 27809.901,E2 27809.901} C_VEL
LIN {X 0,Y 575.909,Z 801.568,A -85,B 0,C 180,E1 27807.811,E2 27807.811} C_VEL
LIN {X 0,Y 575.914,Z 799.024,A -85,B 0,C 180,E1 27805.819,E2 27805.819} C_VEL
LIN {X 0,Y 575.925,Z 794.857,A -85,B 0,C 180,E1 27803.821,E2 27803.821} C_VEL
LIN {X 0,Y 575.955,Z 788.986,A -85,B 0,C 180,E1 27801.816,E2 27801.816} C_VEL
LIN {X 0,Y 575.999,Z 781.322,A -85,B 0,C 180,E1 27799.814,E2 27799.814} C_VEL
LIN {X 0,Y 576.078,Z 771.986,A -85,B 0,C 180,E1 27797.877,E2 27797.877} C_VEL
LIN {X 0,Y 576.198,Z 761.242,A -85,B 0,C 180,E1 27796.043,E2 27796.043} C_VEL
LIN {X 0,Y 576.357,Z 749.105,A -85,B 0,C 180,E1 27794.299,E2 27794.299} C_VEL
LIN {X 0,Y 576.581,Z 734.646,A -85,B 0,C 180,E1 27792.543,E2 27792.543} C_VEL
LIN {X 0,Y 576.853,Z 718.934,A -85,B 0,C 180,E1 27790.93,E2 27790.93} C_VEL
LIN {X 0,Y 577.16,Z 702.009,A -85,B 0,C 180,E1 27789.463,E2 27789.463} C_VEL
LIN {X 0,Y 577.497,Z 683.944,A -85,B 0,C 180,E1 27788.147,E2 27788.147} C_VEL
LIN {X 0,Y 577.839,Z 665.524,A -85,B 0,C 180,E1 27787.029,E2 27787.029} C_VEL
LIN {X 0,Y 578.168,Z 646.388,A -85,B 0,C 180,E1 27786.076,E2 27786.076} C_VEL
LIN {X 0,Y 578.442,Z 626.619,A -85,B 0,C 180,E1 27785.3,E2 27785.3} C_VEL
LIN {X 0,Y 578.659,Z 606.575,A -85,B 0,C 180,E1 27784.707,E2 27784.707} C_VEL
LIN {X 0,Y 578.847,Z 585.728,A -85,B 0,C 180,E1 27784.283,E2 27784.283} C_VEL
LIN {X 0,Y 579.668,Z 334.252,A -85,B 0,C 180,E1 27780.871,E2 27780.871} C_VEL
LIN {X 0,Y 578.707,Z 328.895,A -85,B 0,C 180,E1 27780.729,E2 27780.729} C_VEL
LIN {X 0,Y 579.316,Z 283.626,A -85,B 0,C 180,E1 27777.537,E2 27777.537} C_VEL
LIN {X 0,Y 579.492,Z 265.046,A -85,B 0,C 180,E1 27776.188,E2 27776.188} C_VEL
LIN {X 0,Y 576.198,Z 256.279,A -85,B 0,C 180,E1 27775.279,E2 27775.279} C_VEL
LIN {X 0,Y 576.154,Z 255.963,A -85,B 0,C 180,E1 27774.309,E2 27774.309} C_VEL
LIN {X 0,Y 576.149,Z 255.96,A -85,B 0,C 180,E1 27770.954,E2 27770.954} C_VEL
LIN {X 0,Y 576.139,Z 255.968,A -85,B 0,C 180,E1 27767.672,E2 27767.672} C_VEL
LIN {X 0,Y 576.155,Z 255.963,A -85,B 0,C 180,E1 27764.36,E2 27764.36} C_VEL
LIN {X 0,Y 576.148,Z 255.969,A -85,B 0,C 180,E1 27760.985,E2 27760.985} C_VEL
LIN {X 0,Y 576.147,Z 255.961,A -85,B 0,C 180,E1 27757.778,E2 27757.778} C_VEL
LIN {X 0,Y 576.136,Z 255.966,A -85,B 0,C 180,E1 27754.576,E2 27754.576} C_VEL
LIN {X 0,Y 576.161,Z 255.959,A -85,B 0,C 180,E1 27751.257,E2 27751.257} C_VEL
LIN {X 0,Y 576.158,Z 255.962,A -85,B 0,C 180,E1 27747.941,E2 27747.941} C_VEL
LIN {X 0,Y 576.127,Z 255.968,A -85,B 0,C 180,E1 27744.724,E2 27744.724} C_VEL
LIN {X 0,Y 576.157,Z 255.965,A -85,B 0,C 180,E1 27741.48,E2 27741.48} C_VEL
LIN {X 0,Y 576.123,Z 255.963,A -85,B 0,C 180,E1 27738.308,E2 27738.308} C_VEL
LIN {X 0,Y 576.136,Z 255.967,A -85,B 0,C 180,E1 27734.986,E2 27734.986} C_VEL
LIN {X 0,Y 576.156,Z 255.964,A -85,B 0,C 180,E1 27731.715,E2 27731.715} C_VEL
LIN {X 0,Y 576.107,Z 255.968,A -85,B 0,C 180,E1 27728.484,E2 27728.484} C_VEL
LIN {X 0,Y 576.159,Z 255.967,A -85,B 0,C 180,E1 27725.277,E2 27725.277} C_VEL
LIN {X 0,Y 576.101,Z 255.966,A -85,B 0,C 180,E1 27722.188,E2 27722.188} C_VEL
LIN {X 0,Y 576.12,Z 255.97,A -85,B 0,C 180,E1 27718.906,E2 27718.906} C_VEL
LIN {X 0,Y 576.104,Z 255.967,A -85,B 0,C 180,E1 27715.92,E2 27715.92} C_VEL
LIN {X 0,Y 576.094,Z 255.968,A -85,B 0,C 180,E1 27712.621,E2 27712.621} C_VEL
LIN {X 0,Y 576.121,Z 255.97,A -85,B 0,C 180,E1 27709.602,E2 27709.602} C_VEL
LIN {X 0,Y 576.077,Z 255.971,A -85,B 0,C 180,E1 27706.392,E2 27706.392} C_VEL
LIN {X 0,Y 576.149,Z 255.969,A -85,B 0,C 180,E1 27703.257,E2 27703.257} C_VEL
LIN {X 0,Y 576.078,Z 255.969,A -85,B 0,C 180,E1 27700.112,E2 27700.112} C_VEL
LIN {X 0,Y 576.131,Z 255.968,A -85,B 0,C 180,E1 27696.908,E2 27696.908} C_VEL
LIN {X 0,Y 576.096,Z 255.97,A -85,B 0,C 180,E1 27693.843,E2 27693.843} C_VEL
LIN {X 0,Y 576.102,Z 255.966,A -85,B 0,C 180,E1 27690.469,E2 27690.469} C_VEL
LIN {X 0,Y 576.133,Z 255.964,A -85,B 0,C 180,E1 27687.453,E2 27687.453} C_VEL
LIN {X 0,Y 576.102,Z 255.965,A -85,B 0,C 180,E1 27684.206,E2 27684.206} C_VEL
LIN {X 0,Y 576.162,Z 255.967,A -85,B 0,C 180,E1 27681.026,E2 27681.026} C_VEL
LIN {X 0,Y 576.113,Z 255.962,A -85,B 0,C 180,E1 27677.806,E2 27677.806} C_VEL
LIN {X 0,Y 576.135,Z 255.959,A -85,B 0,C 180,E1 27674.498,E2 27674.498} C_VEL
LIN {X 0,Y 576.155,Z 255.96,A -85,B 0,C 180,E1 27671.257,E2 27671.257} C_VEL
LIN {X 0,Y 576.118,Z 255.942,A -85,B 0,C 180,E1 27668.009,E2 27668.009} C_VEL
LIN {X 0,Y 576.186,Z 256.274,A -85,B 0,C 180,E1 27667.46,E2 27667.46} C_VEL
LIN {X 0,Y 579.91,Z 265.341,A -85,B 0,C 180,E1 27666.539,E2 27666.539} C_VEL
LIN {X 0,Y 580.477,Z 266.77,A -85,B 0,C 180,E1 27666.403,E2 27666.403} C_VEL
LIN {X 0,Y 580.075,Z 302.855,A -85,B 0,C 180,E1 27664.122,E2 27664.122} C_VEL
LIN {X 0,Y 581.015,Z 309.415,A -85,B 0,C 180,E1 27663.962,E2 27663.962} C_VEL
LIN {X 0,Y 580.138,Z 531.902,A -85,B 0,C 180,E1 27660.824,E2 27660.824} C_VEL
LIN {X 0,Y 579.823,Z 609.104,A -85,B 0,C 180,E1 27659.725,E2 27659.725} C_VEL
LIN {X 0,Y 579.566,Z 630.285,A -85,B 0,C 180,E1 27659.237,E2 27659.237} C_VEL
LIN {X 0,Y 579.254,Z 651.775,A -85,B 0,C 180,E1 27658.563,E2 27658.563} C_VEL
LIN {X 0,Y 578.945,Z 672.148,A -85,B 0,C 180,E1 27657.738,E2 27657.738} C_VEL
LIN {X 0,Y 578.526,Z 691.762,A -85,B 0,C 180,E1 27656.757,E2 27656.757} C_VEL
LIN {X 0,Y 578.136,Z 711.729,A -85,B 0,C 180,E1 27655.562,E2 27655.562} C_VEL
LIN {X 0,Y 577.739,Z 730.806,A -85,B 0,C 180,E1 27654.211,E2 27654.211} C_VEL
LIN {X 0,Y 577.327,Z 748.698,A -85,B 0,C 180,E1 27652.718,E2 27652.718} C_VEL
LIN {X 0,Y 576.965,Z 765.835,A -85,B 0,C 180,E1 27651.058,E2 27651.058} C_VEL
LIN {X 0,Y 576.678,Z 781.172,A -85,B 0,C 180,E1 27649.339,E2 27649.339} C_VEL
LIN {X 0,Y 576.446,Z 795.628,A -85,B 0,C 180,E1 27647.461,E2 27647.461} C_VEL
LIN {X 0,Y 576.246,Z 808.472,A -85,B 0,C 180,E1 27645.498,E2 27645.498} C_VEL
LIN {X 0,Y 576.098,Z 819.293,A -85,B 0,C 180,E1 27643.55,E2 27643.55} C_VEL
LIN {X 0,Y 576.012,Z 828.845,A -85,B 0,C 180,E1 27641.514,E2 27641.514} C_VEL
LIN {X 0,Y 575.953,Z 836.531,A -85,B 0,C 180,E1 27639.492,E2 27639.492} C_VEL
LIN {X 0,Y 575.927,Z 843.145,A -85,B 0,C 180,E1 27637.281,E2 27637.281} C_VEL
LIN {X 0,Y 575.918,Z 847.825,A -85,B 0,C 180,E1 27635.179,E2 27635.179} C_VEL
LIN {X 0,Y 575.916,Z 850.784,A -85,B 0,C 180,E1 27633.085,E2 27633.085} C_VEL
LIN {X 0,Y 575.909,Z 852.306,A -85,B 0,C 180,E1 27630.895,E2 27630.895} C_VEL
LIN {X 0,Y 575.911,Z 852.239,A -85,B 0,C 180,E1 27628.806,E2 27628.806} C_VEL
LIN {X 0,Y 575.917,Z 850.559,A -85,B 0,C 180,E1 27626.716,E2 27626.716} C_VEL
LIN {X 0,Y 575.92,Z 847.221,A -85,B 0,C 180,E1 27624.521,E2 27624.521} C_VEL
LIN {X 0,Y 575.927,Z 842.43,A -85,B 0,C 180,E1 27622.437,E2 27622.437} C_VEL
LIN {X 0,Y 575.953,Z 835.821,A -85,B 0,C 180,E1 27620.306,E2 27620.306} C_VEL
LIN {X 0,Y 576.016,Z 827.775,A -85,B 0,C 180,E1 27618.237,E2 27618.237} C_VEL
LIN {X 0,Y 576.107,Z 818.254,A -85,B 0,C 180,E1 27616.245,E2 27616.245} C_VEL
LIN {X 0,Y 576.25,Z 807.192,A -85,B 0,C 180,E1 27614.296,E2 27614.296} C_VEL
LIN {X 0,Y 576.457,Z 794.883,A -85,B 0,C 180,E1 27612.435,E2 27612.435} C_VEL
LIN {X 0,Y 576.698,Z 780.322,A -85,B 0,C 180,E1 27610.557,E2 27610.557} C_VEL
LIN {X 0,Y 576.983,Z 765.174,A -85,B 0,C 180,E1 27608.873,E2 27608.873} C_VEL
LIN {X 0,Y 577.348,Z 747.49,A -85,B 0,C 180,E1 27607.175,E2 27607.175} C_VEL
LIN {X 0,Y 577.747,Z 729.986,A -85,B 0,C 180,E1 27605.728,E2 27605.728} C_VEL
LIN {X 0,Y 578.137,Z 711.731,A -85,B 0,C 180,E1 27604.438,E2 27604.438} C_VEL
LIN {X 0,Y 578.526,Z 691.764,A -85,B 0,C 180,E1 27603.243,E2 27603.243} C_VEL
LIN {X 0,Y 578.945,Z 672.148,A -85,B 0,C 180,E1 27602.262,E2 27602.262} C_VEL
LIN {X 0,Y 579.254,Z 651.779,A -85,B 0,C 180,E1 27601.437,E2 27601.437} C_VEL
LIN {X 0,Y 579.571,Z 629.773,A -85,B 0,C 180,E1 27600.749,E2 27600.749} C_VEL
LIN {X 0,Y 579.83,Z 608.464,A -85,B 0,C 180,E1 27600.265,E2 27600.265} C_VEL
LIN {X 0,Y 580.273,Z 500.04,A -85,B 0,C 180,E1 27598.733,E2 27598.733} C_VEL
LIN {X 0,Y 580.941,Z 307.606,A -85,B 0,C 180,E1 27596.007,E2 27596.007} C_VEL
LIN {X 0,Y 579.978,Z 301.949,A -85,B 0,C 180,E1 27595.842,E2 27595.842} C_VEL
LIN {X 0,Y 580.391,Z 266.355,A -85,B 0,C 180,E1 27593.563,E2 27593.563} C_VEL
LIN {X 0,Y 576.202,Z 256.359,A -85,B 0,C 180,E1 27592.558,E2 27592.558} C_VEL
LIN {X 0,Y 576.118,Z 255.938,A -85,B 0,C 180,E1 27592.095,E2 27592.095} C_VEL
LIN {X 0,Y 576.159,Z 255.959,A -85,B 0,C 180,E1 27588.864,E2 27588.864} C_VEL
LIN {X 0,Y 576.126,Z 255.96,A -85,B 0,C 180,E1 27585.623,E2 27585.623} C_VEL
LIN {X 0,Y 576.12,Z 255.963,A -85,B 0,C 180,E1 27582.328,E2 27582.328} C_VEL
LIN {X 0,Y 576.16,Z 255.965,A -85,B 0,C 180,E1 27579.132,E2 27579.132} C_VEL
LIN {X 0,Y 576.102,Z 255.965,A -85,B 0,C 180,E1 27575.917,E2 27575.917} C_VEL
LIN {X 0,Y 576.148,Z 255.964,A -85,B 0,C 180,E1 27572.664,E2 27572.664} C_VEL
LIN {X 0,Y 576.105,Z 255.966,A -85,B 0,C 180,E1 27569.531,E2 27569.531} C_VEL
LIN {X 0,Y 576.098,Z 255.97,A -85,B 0,C 180,E1 27566.157,E2 27566.157} C_VEL
LIN {X 0,Y 576.131,Z 255.968,A -85,B 0,C 180,E1 27563.092,E2 27563.092} C_VEL
LIN {X 0,Y 576.082,Z 255.968,A -85,B 0,C 180,E1 27559.888,E2 27559.888} C_VEL
LIN {X 0,Y 576.152,Z 255.97,A -85,B 0,C 180,E1 27556.743,E2 27556.743} C_VEL
LIN {X 0,Y 576.075,Z 255.971,A -85,B 0,C 180,E1 27553.607,E2 27553.607} C_VEL
LIN {X 0,Y 576.12,Z 255.97,A -85,B 0,C 180,E1 27550.398,E2 27550.398} C_VEL
LIN {X 0,Y 576.088,Z 255.969,A -85,B 0,C 180,E1 27547.379,E2 27547.379} C_VEL
LIN {X 0,Y 576.096,Z 255.968,A -85,B 0,C 180,E1 27543.981,E2 27543.981} C_VEL
LIN {X 0,Y 576.124,Z 255.97,A -85,B 0,C 180,E1 27540.994,E2 27540.994} C_VEL
LIN {X 0,Y 576.099,Z 255.967,A -85,B 0,C 180,E1 27537.812,E2 27537.812} C_VEL
LIN {X 0,Y 576.156,Z 255.968,A -85,B 0,C 180,E1 27534.723,E2 27534.723} C_VEL
LIN {X 0,Y 576.103,Z 255.968,A -85,B 0,C 180,E1 27531.516,E2 27531.516} C_VEL
LIN {X 0,Y 576.156,Z 255.965,A -85,B 0,C 180,E1 27528.285,E2 27528.285} C_VEL
LIN {X 0,Y 576.122,Z 255.966,A -85,B 0,C 180,E1 27525.116,E2 27525.116} C_VEL
LIN {X 0,Y 576.117,Z 255.968,A -85,B 0,C 180,E1 27523.24,E2 27523.24} C_VEL
LIN {X 0,Y 575.16,Z 256.093,A -85,B 0,C 180,E1 27522.474,E2 27522.474} C_VEL
LIN {X 0,Y 568.646,Z 256.901,A -85,B 0,C 180,E1 27520.268,E2 27520.268} C_VEL
LIN {X 0,Y 568.187,Z 256.954,A -85,B 0,C 180,E1 27519.764,E2 27519.764} C_VEL
LIN {X 0,Y 568.221,Z 256.958,A -85,B 0,C 180,E1 27516.567,E2 27516.567} C_VEL
LIN {X 0,Y 568.185,Z 256.953,A -85,B 0,C 180,E1 27513.337,E2 27513.337} C_VEL
LIN {X 0,Y 568.224,Z 256.944,A -85,B 0,C 180,E1 27510.018,E2 27510.018} C_VEL
LIN {X 0,Y 568.215,Z 256.956,A -85,B 0,C 180,E1 27506.7,E2 27506.7} C_VEL
LIN {X 0,Y 568.194,Z 256.95,A -85,B 0,C 180,E1 27503.36,E2 27503.36} C_VEL
LIN {X 0,Y 568.212,Z 256.953,A -85,B 0,C 180,E1 27500.102,E2 27500.102} C_VEL
LIN {X 0,Y 568.216,Z 256.95,A -85,B 0,C 180,E1 27496.758,E2 27496.758} C_VEL
LIN {X 0,Y 568.205,Z 256.947,A -85,B 0,C 180,E1 27493.385,E2 27493.385} C_VEL
LIN {X 0,Y 568.201,Z 256.947,A -85,B 0,C 180,E1 27490.208,E2 27490.208} C_VEL
LIN {X 0,Y 568.209,Z 256.949,A -85,B 0,C 180,E1 27486.976,E2 27486.976} C_VEL
LIN {X 0,Y 568.25,Z 257.243,A -85,B 0,C 180,E1 27485.124,E2 27485.124} C_VEL
LIN {X 0,Y 570.526,Z 263.325,A -85,B 0,C 180,E1 27484.456,E2 27484.456} C_VEL
LIN {X 0,Y 572.512,Z 268.967,A -85,B 0,C 180,E1 27483.896,E2 27483.896} C_VEL
LIN {X 0,Y 571.705,Z 314.077,A -85,B 0,C 180,E1 27480.631,E2 27480.631} C_VEL
LIN {X 0,Y 571.541,Z 329.554,A -85,B 0,C 180,E1 27479.564,E2 27479.564} C_VEL
LIN {X 0,Y 572.69,Z 337.046,A -85,B 0,C 180,E1 27479.389,E2 27479.389} C_VEL
LIN {X 0,Y 571.614,Z 590.327,A -85,B 0,C 180,E1 27475.901,E2 27475.901} C_VEL
LIN {X 0,Y 571.362,Z 610.632,A -85,B 0,C 180,E1 27475.44,E2 27475.44} C_VEL
LIN {X 0,Y 571.036,Z 630.846,A -85,B 0,C 180,E1 27474.793,E2 27474.793} C_VEL
LIN {X 0,Y 570.68,Z 650.206,A -85,B 0,C 180,E1 27473.983,E2 27473.983} C_VEL
LIN {X 0,Y 570.302,Z 668.879,A -85,B 0,C 180,E1 27473.01,E2 27473.01} C_VEL
LIN {X 0,Y 569.881,Z 687.408,A -85,B 0,C 180,E1 27471.836,E2 27471.836} C_VEL
LIN {X 0,Y 569.453,Z 704.875,A -85,B 0,C 180,E1 27470.504,E2 27470.504} C_VEL
LIN {X 0,Y 569.077,Z 721.049,A -85,B 0,C 180,E1 27469.045,E2 27469.045} C_VEL
LIN {X 0,Y 568.752,Z 735.705,A -85,B 0,C 180,E1 27467.494,E2 27467.494} C_VEL
LIN {X 0,Y 568.487,Z 749.212,A -85,B 0,C 180,E1 27465.819,E2 27465.819} C_VEL
LIN {X 0,Y 568.267,Z 761.965,A -85,B 0,C 180,E1 27463.948,E2 27463.948} C_VEL
LIN {X 0,Y 568.116,Z 772.569,A -85,B 0,C 180,E1 27462.089,E2 27462.089} C_VEL
LIN {X 0,Y 568.018,Z 781.757,A -85,B 0,C 180,E1 27460.138,E2 27460.138} C_VEL
LIN {X 0,Y 567.961,Z 789.378,A -85,B 0,C 180,E1 27458.096,E2 27458.096} C_VEL
LIN {X 0,Y 567.93,Z 795.138,A -85,B 0,C 180,E1 27456.063,E2 27456.063} C_VEL
LIN {X 0,Y 567.918,Z 799.199,A -85,B 0,C 180,E1 27454.038,E2 27454.038} C_VEL
LIN {X 0,Y 567.915,Z 801.642,A -85,B 0,C 180,E1 27452.018,E2 27452.018} C_VEL
LIN {X 0,Y 567.914,Z 802.493,A -85,B 0,C 180,E1 27449.899,E2 27449.899} C_VEL
LIN {X 0,Y 567.908,Z 801.567,A -85,B 0,C 180,E1 27447.78,E2 27447.78} C_VEL
LIN {X 0,Y 567.913,Z 799.023,A -85,B 0,C 180,E1 27445.76,E2 27445.76} C_VEL
LIN {X 0,Y 567.926,Z 794.856,A -85,B 0,C 180,E1 27443.734,E2 27443.734} C_VEL
LIN {X 0,Y 567.962,Z 788.984,A -85,B 0,C 180,E1 27441.7,E2 27441.7} C_VEL
LIN {X 0,Y 568.023,Z 781.584,A -85,B 0,C 180,E1 27439.73,E2 27439.73} C_VEL
LIN {X 0,Y 568.12,Z 772.502,A -85,B 0,C 180,E1 27437.808,E2 27437.808} C_VEL
LIN {X 0,Y 568.27,Z 761.879,A -85,B 0,C 180,E1 27435.948,E2 27435.948} C_VEL
LIN {X 0,Y 568.474,Z 749.829,A -85,B 0,C 180,E1 27434.174,E2 27434.174} C_VEL
LIN {X 0,Y 568.734,Z 736.494,A -85,B 0,C 180,E1 27432.505,E2 27432.505} C_VEL
LIN {X 0,Y 569.064,Z 721.69,A -85,B 0,C 180,E1 27430.926,E2 27430.926} C_VEL
LIN {X 0,Y 569.45,Z 705.325,A -85,B 0,C 180,E1 27429.442,E2 27429.442} C_VEL
LIN {X 0,Y 569.868,Z 687.9,A -85,B 0,C 180,E1 27428.11,E2 27428.11} C_VEL
LIN {X 0,Y 570.262,Z 670.297,A -85,B 0,C 180,E1 27426.984,E2 27426.984} C_VEL
LIN {X 0,Y 570.664,Z 650.933,A -85,B 0,C 180,E1 27425.961,E2 27425.961} C_VEL
LIN {X 0,Y 571.033,Z 630.98,A -85,B 0,C 180,E1 27425.122,E2 27425.122} C_VEL
LIN {X 0,Y 571.362,Z 610.688,A -85,B 0,C 180,E1 27424.471,E2 27424.471} C_VEL
LIN {X 0,Y 571.614,Z 590.294,A -85,B 0,C 180,E1 27424.008,E2 27424.008} C_VEL
LIN {X 0,Y 572.682,Z 335.647,A -85,B 0,C 180,E1 27420.501,E2 27420.501} C_VEL
LIN {X 0,Y 571.46,Z 328.894,A -85,B 0,C 180,E1 27420.321,E2 27420.321} C_VEL
LIN {X 0,Y 572.241,Z 283.615,A -85,B 0,C 180,E1 27417.086,E2 27417.086} C_VEL
LIN {X 0,Y 572.469,Z 268.428,A -85,B 0,C 180,E1 27415.971,E2 27415.971} C_VEL
LIN {X 0,Y 568.279,Z 257.393,A -85,B 0,C 180,E1 27414.816,E2 27414.816} C_VEL
LIN {X 0,Y 568.212,Z 256.949,A -85,B 0,C 180,E1 27414.254,E2 27414.254} C_VEL
LIN {X 0,Y 568.209,Z 256.946,A -85,B 0,C 180,E1 27410.897,E2 27410.897} C_VEL
LIN {X 0,Y 568.202,Z 256.958,A -85,B 0,C 180,E1 27407.628,E2 27407.628} C_VEL
LIN {X 0,Y 568.219,Z 256.952,A -85,B 0,C 180,E1 27404.262,E2 27404.262} C_VEL
LIN {X 0,Y 568.205,Z 256.957,A -85,B 0,C 180,E1 27400.89,E2 27400.89} C_VEL
LIN {X 0,Y 568.208,Z 256.951,A -85,B 0,C 180,E1 27397.634,E2 27397.634} C_VEL
LIN {X 0,Y 568.202,Z 256.953,A -85,B 0,C 180,E1 27394.384,E2 27394.384} C_VEL
LIN {X 0,Y 568.206,Z 256.948,A -85,B 0,C 180,E1 27391.026,E2 27391.026} C_VEL
LIN {X 0,Y 568.215,Z 256.954,A -85,B 0,C 180,E1 27387.681,E2 27387.681} C_VEL
LIN {X 0,Y 568.189,Z 256.954,A -85,B 0,C 180,E1 27384.427,E2 27384.427} C_VEL
LIN {X 0,Y 568.213,Z 256.96,A -85,B 0,C 180,E1 27381.145,E2 27381.145} C_VEL
LIN {X 0,Y 568.216,Z 256.949,A -85,B 0,C 180,E1 27377.829,E2 27377.829} C_VEL
LIN {X 0,Y 568.177,Z 256.953,A -85,B 0,C 180,E1 27374.569,E2 27374.569} C_VEL
LIN {X 0,Y 568.222,Z 256.958,A -85,B 0,C 180,E1 27371.366,E2 27371.366} C_VEL
LIN {X 0,Y 568.173,Z 256.956,A -85,B 0,C 180,E1 27368.195,E2 27368.195} C_VEL
LIN {X 0,Y 568.18,Z 256.959,A -85,B 0,C 180,E1 27364.846,E2 27364.846} C_VEL
LIN {X 0,Y 568.198,Z 256.953,A -85,B 0,C 180,E1 27361.714,E2 27361.714} C_VEL
LIN {X 0,Y 568.156,Z 256.958,A -85,B 0,C 180,E1 27358.488,E2 27358.488} C_VEL
LIN {X 0,Y 568.219,Z 256.957,A -85,B 0,C 180,E1 27355.357,E2 27355.357} C_VEL
LIN {X 0,Y 568.146,Z 256.956,A -85,B 0,C 180,E1 27352.211,E2 27352.211} C_VEL
LIN {X 0,Y 568.191,Z 256.957,A -85,B 0,C 180,E1 27349.045,E2 27349.045} C_VEL
LIN {X 0,Y 568.14,Z 256.96,A -85,B 0,C 180,E1 27346.049,E2 27346.049} C_VEL
LIN {X 0,Y 568.163,Z 256.96,A -85,B 0,C 180,E1 27342.804,E2 27342.804} C_VEL
LIN {X 0,Y 568.152,Z 256.957,A -85,B 0,C 180,E1 27339.823,E2 27339.823} C_VEL
LIN {X 0,Y 568.152,Z 256.958,A -85,B 0,C 180,E1 27336.454,E2 27336.454} C_VEL
LIN {X 0,Y 568.207,Z 256.957,A -85,B 0,C 180,E1 27333.339,E2 27333.339} C_VEL
LIN {X 0,Y 568.155,Z 256.955,A -85,B 0,C 180,E1 27330.178,E2 27330.178} C_VEL
LIN {X 0,Y 568.216,Z 256.957,A -85,B 0,C 180,E1 27326.942,E2 27326.942} C_VEL
LIN {X 0,Y 568.171,Z 256.955,A -85,B 0,C 180,E1 27323.752,E2 27323.752} C_VEL
LIN {X 0,Y 568.181,Z 256.956,A -85,B 0,C 180,E1 27320.421,E2 27320.421} C_VEL
LIN {X 0,Y 568.219,Z 256.954,A -85,B 0,C 180,E1 27317.201,E2 27317.201} C_VEL
LIN {X 0,Y 568.176,Z 256.95,A -85,B 0,C 180,E1 27313.967,E2 27313.967} C_VEL
LIN {X 0,Y 568.223,Z 256.945,A -85,B 0,C 180,E1 27310.677,E2 27310.677} C_VEL
LIN {X 0,Y 568.215,Z 257.182,A -85,B 0,C 180,E1 27308.03,E2 27308.03} C_VEL
LIN {X 0,Y 569.524,Z 260.471,A -85,B 0,C 180,E1 27307.648,E2 27307.648} C_VEL
LIN {X 0,Y 573.639,Z 270.585,A -85,B 0,C 180,E1 27306.653,E2 27306.653} C_VEL
LIN {X 0,Y 573.098,Z 302.318,A -85,B 0,C 180,E1 27304.61,E2 27304.61} C_VEL
LIN {X 0,Y 574.37,Z 310.696,A -85,B 0,C 180,E1 27304.391,E2 27304.391} C_VEL
LIN {X 0,Y 573.263,Z 532.792,A -85,B 0,C 180,E1 27301.222,E2 27301.222} C_VEL
LIN {X 0,Y 572.869,Z 609.208,A -85,B 0,C 180,E1 27300.121,E2 27300.121} C_VEL
LIN {X 0,Y 572.543,Z 630.545,A -85,B 0,C 180,E1 27299.624,E2 27299.624} C_VEL
LIN {X 0,Y 572.143,Z 652.603,A -85,B 0,C 180,E1 27298.919,E2 27298.919} C_VEL
LIN {X 0,Y 571.743,Z 673.408,A -85,B 0,C 180,E1 27298.061,E2 27298.061} C_VEL
LIN {X 0,Y 571.222,Z 692.759,A -85,B 0,C 180,E1 27297.071,E2 27297.071} C_VEL
LIN {X 0,Y 570.705,Z 713.161,A -85,B 0,C 180,E1 27295.821,E2 27295.821} C_VEL
LIN {X 0,Y 570.201,Z 732.126,A -85,B 0,C 180,E1 27294.445,E2 27294.445} C_VEL
LIN {X 0,Y 569.698,Z 749.906,A -85,B 0,C 180,E1 27292.93,E2 27292.93} C_VEL
LIN {X 0,Y 569.254,Z 766.542,A -85,B 0,C 180,E1 27291.282,E2 27291.282} C_VEL
LIN {X 0,Y 568.878,Z 782.023,A -85,B 0,C 180,E1 27289.508,E2 27289.508} C_VEL
LIN {X 0,Y 568.58,Z 796.273,A -85,B 0,C 180,E1 27287.615,E2 27287.615} C_VEL
LIN {X 0,Y 568.33,Z 809.105,A -85,B 0,C 180,E1 27285.615,E2 27285.615} C_VEL
LIN {X 0,Y 568.148,Z 819.814,A -85,B 0,C 180,E1 27283.64,E2 27283.64} C_VEL
LIN {X 0,Y 568.036,Z 829.253,A -85,B 0,C 180,E1 27281.575,E2 27281.575} C_VEL
LIN {X 0,Y 567.965,Z 836.885,A -85,B 0,C 180,E1 27279.525,E2 27279.525} C_VEL
LIN {X 0,Y 567.928,Z 843.145,A -85,B 0,C 180,E1 27277.384,E2 27277.384} C_VEL
LIN {X 0,Y 567.919,Z 847.825,A -85,B 0,C 180,E1 27275.253,E2 27275.253} C_VEL
LIN {X 0,Y 567.916,Z 850.784,A -85,B 0,C 180,E1 27273.129,E2 27273.129} C_VEL
LIN {X 0,Y 567.91,Z 852.306,A -85,B 0,C 180,E1 27270.908,E2 27270.908} C_VEL
LIN {X 0,Y 567.91,Z 852.239,A -85,B 0,C 180,E1 27268.789,E2 27268.789} C_VEL
LIN {X 0,Y 567.915,Z 850.487,A -85,B 0,C 180,E1 27266.605,E2 27266.605} C_VEL
LIN {X 0,Y 567.92,Z 847.015,A -85,B 0,C 180,E1 27264.342,E2 27264.342} C_VEL
LIN {X 0,Y 567.941,Z 842.128,A -85,B 0,C 180,E1 27262.209,E2 27262.209} C_VEL
LIN {X 0,Y 567.97,Z 835.821,A -85,B 0,C 180,E1 27260.168,E2 27260.168} C_VEL
LIN {X 0,Y 568.048,Z 827.981,A -85,B 0,C 180,E1 27258.116,E2 27258.116} C_VEL
LIN {X 0,Y 568.16,Z 818.775,A -85,B 0,C 180,E1 27256.153,E2 27256.153} C_VEL
LIN {X 0,Y 568.348,Z 807.193,A -85,B 0,C 180,E1 27254.072,E2 27254.072} C_VEL
LIN {X 0,Y 568.607,Z 794.881,A -85,B 0,C 180,E1 27252.184,E2 27252.184} C_VEL
LIN {X 0,Y 568.928,Z 780.323,A -85,B 0,C 180,E1 27250.28,E2 27250.28} C_VEL
LIN {X 0,Y 569.299,Z 765.091,A -85,B 0,C 180,E1 27248.565,E2 27248.565} C_VEL
LIN {X 0,Y 569.759,Z 747.491,A -85,B 0,C 180,E1 27246.854,E2 27246.854} C_VEL
LIN {X 0,Y 570.245,Z 730.034,A -85,B 0,C 180,E1 27245.391,E2 27245.391} C_VEL
LIN {X 0,Y 570.753,Z 711.728,A -85,B 0,C 180,E1 27244.083,E2 27244.083} C_VEL
LIN {X 0,Y 571.248,Z 691.767,A -85,B 0,C 180,E1 27242.874,E2 27242.874} C_VEL
LIN {X 0,Y 571.759,Z 672.152,A -85,B 0,C 180,E1 27241.883,E2 27241.883} C_VEL
LIN {X 0,Y 572.169,Z 651.777,A -85,B 0,C 180,E1 27241.05,E2 27241.05} C_VEL
LIN {X 0,Y 572.551,Z 629.775,A -85,B 0,C 180,E1 27240.355,E2 27240.355} C_VEL
LIN {X 0,Y 572.877,Z 608.357,A -85,B 0,C 180,E1 27239.865,E2 27239.865} C_VEL
LIN {X 0,Y 573.541,Z 476.428,A -85,B 0,C 180,E1 27237.983,E2 27237.983} C_VEL
LIN {X 0,Y 574.239,Z 308.727,A -85,B 0,C 180,E1 27235.571,E2 27235.571} C_VEL
LIN {X 0,Y 573.072,Z 301.841,A -85,B 0,C 180,E1 27235.366,E2 27235.366} C_VEL
LIN {X 0,Y 573.601,Z 270.006,A -85,B 0,C 180,E1 27233.306,E2 27233.306} C_VEL
LIN {X 0,Y 568.259,Z 257.433,A -85,B 0,C 180,E1 27232.023,E2 27232.023} C_VEL
LIN {X 0,Y 568.19,Z 256.929,A -85,B 0,C 180,E1 27231.705,E2 27231.705} C_VEL
LIN {X 0,Y 568.185,Z 256.956,A -85,B 0,C 180,E1 27228.305,E2 27228.305} C_VEL
LIN {X 0,Y 568.221,Z 256.946,A -85,B 0,C 180,E1 27225.021,E2 27225.021} C_VEL
LIN {X 0,Y 568.172,Z 256.948,A -85,B 0,C 180,E1 27221.832,E2 27221.832} C_VEL
LIN {X 0,Y 568.197,Z 256.956,A -85,B 0,C 180,E1 27218.531,E2 27218.531} C_VEL
LIN {X 0,Y 568.189,Z 256.952,A -85,B 0,C 180,E1 27215.377,E2 27215.377} C_VEL
LIN {X 0,Y 568.162,Z 256.95,A -85,B 0,C 180,E1 27212.104,E2 27212.104} C_VEL
LIN {X 0,Y 568.218,Z 256.954,A -85,B 0,C 180,E1 27208.94,E2 27208.94} C_VEL
LIN {X 0,Y 568.15,Z 256.958,A -85,B 0,C 180,E1 27205.765,E2 27205.765} C_VEL
LIN {X 0,Y 568.196,Z 256.96,A -85,B 0,C 180,E1 27202.558,E2 27202.558} C_VEL
LIN {X 0,Y 568.147,Z 256.956,A -85,B 0,C 180,E1 27199.534,E2 27199.534} C_VEL
LIN {X 0,Y 568.158,Z 256.957,A -85,B 0,C 180,E1 27196.249,E2 27196.249} C_VEL
LIN {X 0,Y 568.156,Z 256.96,A -85,B 0,C 180,E1 27193.225,E2 27193.225} C_VEL
LIN {X 0,Y 568.144,Z 256.96,A -85,B 0,C 180,E1 27189.931,E2 27189.931} C_VEL
LIN {X 0,Y 568.211,Z 256.956,A -85,B 0,C 180,E1 27186.771,E2 27186.771} C_VEL
LIN {X 0,Y 568.148,Z 256.957,A -85,B 0,C 180,E1 27183.632,E2 27183.632} C_VEL
LIN {X 0,Y 568.22,Z 256.956,A -85,B 0,C 180,E1 27180.504,E2 27180.504} C_VEL
LIN {X 0,Y 568.16,Z 256.957,A -85,B 0,C 180,E1 27177.377,E2 27177.377} C_VEL
LIN {X 0,Y 568.181,Z 256.952,A -85,B 0,C 180,E1 27174.04,E2 27174.04} C_VEL
LIN {X 0,Y 568.201,Z 256.96,A -85,B 0,C 180,E1 27170.887,E2 27170.887} C_VEL
LIN {X 0,Y 568.167,Z 256.957,A -85,B 0,C 180,E1 27167.596,E2 27167.596} C_VEL
LIN {X 0,Y 568.223,Z 256.954,A -85,B 0,C 180,E1 27164.382,E2 27164.382} C_VEL
LIN {X 0,Y 568.187,Z 256.955,A -85,B 0,C 180,E1 27161.107,E2 27161.107} C_VEL
LIN {X 0,Y 568.187,Z 256.954,A -85,B 0,C 180,E1 27159.764,E2 27159.764} C_VEL
LIN {X 0,Y 567.179,Z 257.086,A -85,B 0,C 180,E1 27158.987,E2 27158.987} C_VEL
LIN {X 0,Y 560.805,Z 257.881,A -85,B 0,C 180,E1 27156.806,E2 27156.806} C_VEL
LIN {X 0,Y 560.28,Z 257.942,A -85,B 0,C 180,E1 27156.239,E2 27156.239} C_VEL
LIN {X 0,Y 560.264,Z 257.944,A -85,B 0,C 180,E1 27152.93,E2 27152.93} C_VEL
LIN {X 0,Y 560.252,Z 257.935,A -85,B 0,C 180,E1 27149.538,E2 27149.538} C_VEL
LIN {X 0,Y 560.276,Z 257.944,A -85,B 0,C 180,E1 27146.263,E2 27146.263} C_VEL
LIN {X 0,Y 560.268,Z 257.936,A -85,B 0,C 180,E1 27142.9,E2 27142.9} C_VEL
LIN {X 0,Y 560.264,Z 257.942,A -85,B 0,C 180,E1 27139.484,E2 27139.484} C_VEL
LIN {X 0,Y 560.27,Z 257.944,A -85,B 0,C 180,E1 27136.177,E2 27136.177} C_VEL
LIN {X 0,Y 560.274,Z 257.936,A -85,B 0,C 180,E1 27132.822,E2 27132.822} C_VEL
LIN {X 0,Y 560.271,Z 257.931,A -85,B 0,C 180,E1 27129.4,E2 27129.4} C_VEL
LIN {X 0,Y 560.26,Z 257.933,A -85,B 0,C 180,E1 27126.08,E2 27126.08} C_VEL
LIN {X 0,Y 560.349,Z 258.39,A -85,B 0,C 180,E1 27125.616,E2 27125.616} C_VEL
LIN {X 0,Y 565.461,Z 271.909,A -85,B 0,C 180,E1 27124.154,E2 27124.154} C_VEL
LIN {X 0,Y 564.499,Z 316.244,A -85,B 0,C 180,E1 27120.907,E2 27120.907} C_VEL
LIN {X 0,Y 564.32,Z 329.538,A -85,B 0,C 180,E1 27119.983,E2 27119.983} C_VEL
LIN {X 0,Y 565.715,Z 338.42,A -85,B 0,C 180,E1 27119.768,E2 27119.768} C_VEL
LIN {X 0,Y 564.417,Z 590.156,A -85,B 0,C 180,E1 27116.26,E2 27116.26} C_VEL
LIN {X 0,Y 564.115,Z 610.506,A -85,B 0,C 180,E1 27115.795,E2 27115.795} C_VEL
LIN {X 0,Y 563.722,Z 630.865,A -85,B 0,C 180,E1 27115.137,E2 27115.137} C_VEL
LIN {X 0,Y 563.296,Z 650.218,A -85,B 0,C 180,E1 27114.317,E2 27114.317} C_VEL
LIN {X 0,Y 562.83,Z 668.822,A -85,B 0,C 180,E1 27113.337,E2 27113.337} C_VEL
LIN {X 0,Y 562.317,Z 687.417,A -85,B 0,C 180,E1 27112.145,E2 27112.145} C_VEL
LIN {X 0,Y 561.805,Z 704.886,A -85,B 0,C 180,E1 27110.796,E2 27110.796} C_VEL
LIN {X 0,Y 561.357,Z 720.761,A -85,B 0,C 180,E1 27109.347,E2 27109.347} C_VEL
LIN {X 0,Y 560.955,Z 735.71,A -85,B 0,C 180,E1 27107.745,E2 27107.745} C_VEL
LIN {X 0,Y 560.615,Z 749.642,A -85,B 0,C 180,E1 27105.99,E2 27105.99} C_VEL
LIN {X 0,Y 560.352,Z 761.97,A -85,B 0,C 180,E1 27104.149,E2 27104.149} C_VEL
LIN {X 0,Y 560.171,Z 772.573,A -85,B 0,C 180,E1 27102.263,E2 27102.263} C_VEL
LIN {X 0,Y 560.046,Z 781.76,A -85,B 0,C 180,E1 27100.284,E2 27100.284} C_VEL
LIN {X 0,Y 559.975,Z 789.38,A -85,B 0,C 180,E1 27098.212,E2 27098.212} C_VEL
LIN {X 0,Y 559.932,Z 795.14,A -85,B 0,C 180,E1 27096.15,E2 27096.15} C_VEL
LIN {X 0,Y 559.918,Z 799.201,A -85,B 0,C 180,E1 27094.096,E2 27094.096} C_VEL
LIN {X 0,Y 559.915,Z 801.641,A -85,B 0,C 180,E1 27092.047,E2 27092.047} C_VEL
LIN {X 0,Y 559.913,Z 802.495,A -85,B 0,C 180,E1 27090,E2 27090} C_VEL
LIN {X 0,Y 559.911,Z 801.634,A -85,B 0,C 180,E1 27087.851,E2 27087.851} C_VEL
LIN {X 0,Y 559.914,Z 799.181,A -85,B 0,C 180,E1 27085.801,E2 27085.801} C_VEL
LIN {X 0,Y 559.928,Z 794.855,A -85,B 0,C 180,E1 27083.644,E2 27083.644} C_VEL
LIN {X 0,Y 559.972,Z 788.982,A -85,B 0,C 180,E1 27081.581,E2 27081.581} C_VEL
LIN {X 0,Y 560.05,Z 781.704,A -85,B 0,C 180,E1 27079.612,E2 27079.612} C_VEL
LIN {X 0,Y 560.173,Z 772.499,A -85,B 0,C 180,E1 27077.632,E2 27077.632} C_VEL
LIN {X 0,Y 560.357,Z 761.876,A -85,B 0,C 180,E1 27075.745,E2 27075.745} C_VEL
LIN {X 0,Y 560.609,Z 749.873,A -85,B 0,C 180,E1 27073.952,E2 27073.952} C_VEL
LIN {X 0,Y 560.934,Z 736.488,A -85,B 0,C 180,E1 27072.254,E2 27072.254} C_VEL
LIN {X 0,Y 561.331,Z 721.684,A -85,B 0,C 180,E1 27070.652,E2 27070.652} C_VEL
LIN {X 0,Y 561.802,Z 705.034,A -85,B 0,C 180,E1 27069.126,E2 27069.126} C_VEL
LIN {X 0,Y 562.322,Z 687.137,A -85,B 0,C 180,E1 27067.745,E2 27067.745} C_VEL
LIN {X 0,Y 562.839,Z 668.476,A -85,B 0,C 180,E1 27066.552,E2 27066.552} C_VEL
LIN {X 0,Y 563.309,Z 649.781,A -85,B 0,C 180,E1 27065.572,E2 27065.572} C_VEL
LIN {X 0,Y 563.749,Z 629.635,A -85,B 0,C 180,E1 27064.727,E2 27064.727} C_VEL
